// TIA Portal project "Laptrinhnangcaocuoiki_V16" (V16)

(* hardware
DEVICE "S7-1200 station_1"  S7-1200 Station
   slot 0: "Rack_0"  S7-1200 Rack  Rack  V1.0
   slot 1: "PLC_1"  CPU 1214C DC/DC/Rly  6ES7 214-1HG40-0XB0  V4.2
DEVICE "PC-System_1"  SIMATIC PC station
   slot 0: "SIMATIC PC station"  Rail  SIMATIC PC-Station  V1.0
      slot 125: "Stationmanager"  Station_Manager  V6.0.4
   slot 1: "HMI_RT_1"  WinCC RT Advanced  6AV2 104-0xxxx-xxxx  15.0.0.0
      slot 33792: "Host interface"  Host interface
   slot 2: "IE general_1"  IE General  IE_CP  V8.2.0
*)

// ===== PLC "PLC_1"  CPU 1214C DC/DC/Rly =====

VAR_GLOBAL   // PLC tag table "Default tag table"
   "Clock_Byte" AT %MB100 : Byte;
   "Clock_10Hz" AT %M100.0 : Bool;
   "Clock_5Hz" AT %M100.1 : Bool;
   "Clock_2.5Hz" AT %M100.2 : Bool;
   "Clock_2Hz" AT %M100.3 : Bool;
   "Clock_1.25Hz" AT %M100.4 : Bool;
   "Clock_1Hz" AT %M100.5 : Bool;
   "Clock_0.625Hz" AT %M100.6 : Bool;
   "Clock_0.5Hz" AT %M100.7 : Bool;
   "Tag_6" AT %M20.0 : Bool;
   "Tag_7" AT %M20.1 : Bool;
   "Tag_14" AT %M20.2 : Bool;
   "Tag_17" AT %M20.3 : Bool;
   "Tag_18" AT %M20.4 : Bool;
   "Tag_24" AT %M20.5 : Bool;
   "Tag_32" AT %M20.6 : Bool;
   "Tag_33" AT %M20.7 : Bool;
   "Tag_34" AT %M21.0 : Bool;
   "Tag_35" AT %M21.1 : Bool;
   "Tag_1" AT %M21.2 : Bool;
   "Tag_36" AT %M21.3 : Bool;
   "Tag_37" AT %M21.4 : Bool;
   "Tag_38" AT %M21.5 : Bool;
   "Tag_39" AT %M21.6 : Bool;
   "Tag_40" AT %M21.7 : Bool;
   "Tag_41" AT %M22.0 : Bool;
   "Tag_42" AT %M22.2 : Bool;
   "Tag_43" AT %M22.1 : Bool;
   "Tag_44" AT %M22.3 : Bool;
   "Tag_45" AT %M22.4 : Bool;
   "Tag_46" AT %M22.5 : Bool;
   "Tag_47" AT %M22.6 : Bool;
   "Tag_48" AT %M22.7 : Bool;
   "Tag_49" AT %M23.0 : Bool;
   "Tag_50" AT %M23.1 : Bool;
   "Tag_51" AT %M23.2 : Bool;
   "Tag_52" AT %M23.3 : Bool;
   "Tag_53" AT %M23.4 : Bool;
   "Tag_54" AT %M23.5 : Bool;
   "Tag_55" AT %M23.6 : Bool;
   "Tag_56" AT %M23.7 : Bool;
   "Tag_57" AT %M24.0 : Bool;
   "Tag_58" AT %M24.1 : Bool;
   "Tag_59" AT %M24.2 : Bool;
   "Tag_2" AT %M24.3 : Bool;
   "Tag_3" AT %M24.4 : Bool;
   "Tag_4" AT %M24.5 : Bool;
   "Tag_5" AT %M24.6 : Bool;
   "Tag_8" AT %M24.7 : Bool;
   "Tag_9" AT %M25.0 : Bool;
   "Tag_10" AT %M25.1 : Bool;
   "Tag_11" AT %M25.2 : Bool;
   "Tag_12" AT %M25.3 : Bool;
   "Tag_13" AT %M25.4 : Bool;
   "Tag_15" AT %M25.5 : Bool;
   "Tag_16" AT %M25.6 : Bool;
   "Tag_19" AT %M25.7 : Bool;
   "Tag_20" AT %M26.0 : Bool;
   "Tag_21" AT %M26.1 : Bool;
   "Tag_22" AT %M26.2 : Bool;
   "Tag_23" AT %M26.3 : Bool;
   "Tag_25" AT %M26.4 : Bool;
   "Tag_26" AT %M26.5 : Bool;
   "Tag_27" AT %M26.6 : Bool;
   "Tag_28" AT %M26.7 : Bool;
   "Tag_29" AT %M27.0 : Bool;
   "Tag_30" AT %M27.1 : Bool;
   "Tag_31" AT %M27.2 : Bool;
   "Tag_60" AT %M27.3 : Bool;
   "Tag_61" AT %M27.4 : Bool;
   "Tag_62" AT %M27.5 : Bool;
   "Tag_63" AT %M27.7 : Bool;
   "Tag_64" AT %M27.6 : Bool;
   "Tag_65" AT %M28.0 : Bool;
   "Tag_66" AT %M28.1 : Bool;
   "Tag_67" AT %M28.2 : Bool;
   "Tag_68" AT %M28.3 : Bool;
   "Tag_69" AT %M28.4 : Bool;
   "Tag_70" AT %M28.5 : Bool;
   "Tag_71" AT %M28.6 : Bool;
   "Tag_72" AT %M28.7 : Bool;
   "Tag_73" AT %M29.0 : Bool;
   "Tag_74" AT %M29.1 : Bool;
   "Tag_75" AT %M29.2 : Bool;
   "Tag_76" AT %M29.3 : Bool;
   "Tag_77" AT %M29.4 : Bool;
   "Tag_78" AT %M29.5 : Bool;
   "Tag_79" AT %M29.6 : Bool;
   "Tag_80" AT %M29.7 : Bool;
   "Tag_81" AT %M30.1 : Bool;
   "Tag_82" AT %M30.2 : Bool;
   "Tag_83" AT %M30.0 : Bool;
   "Tag_84" AT %M30.3 : Bool;
   "Tag_85" AT %M30.4 : Bool;
   "Tag_86" AT %M30.5 : Bool;
   "Tag_87" AT %M30.6 : Bool;
   "Tag_88" AT %M30.7 : Bool;
   "Tag_89" AT %M31.0 : Bool;
   "Tag_90" AT %M31.1 : Bool;
   "Tag_91" AT %M31.2 : Bool;
END_VAR

VAR_GLOBAL   // PLC tag table "M_tag"
   "mStart" AT %M0.0 : Bool;
   "mStop" AT %M0.1 : Bool;
   "mControlOn" AT %M0.2 : Bool;
   "mEnableXiloRice" AT %M0.3 : Bool;
   "mEnableXiloCorn" AT %M0.6 : Bool;
   "mEnableXiloCassava" AT %M1.2 : Bool;
   "mEnableXiloBean" AT %M1.4 : Bool;
   "mEnableXiloFish" AT %M1.7 : Bool;
   "mEnablePourToScale1" AT %M2.6 : Bool;
   "mEnableInverter1_10Hz" AT %M2.7 : Bool;
   "mEnableInverter1_5Hz" AT %M3.0 : Bool;
   "mEnableInverter1_1Hz" AT %M3.1 : Bool;
   "mEnableXiloRice1" AT %M0.4 : Bool;
   "mEnableXiloRice2" AT %M0.5 : Bool;
   "mEnableXiloRice3" AT %M0.7 : Bool;
   "mEnableXiloCorn4" AT %M1.0 : Bool;
   "mEnableXiloCorn5" AT %M1.1 : Bool;
   "mEnableXiloCorn6" AT %M1.3 : Bool;
   "mEnableXiloCorn7" AT %M1.5 : Bool;
   "mEnableXiloCassava8" AT %M1.6 : Bool;
   "mEnableXiloCassava9" AT %M2.0 : Bool;
   "mEnablePourToScale2" AT %M3.2 : Bool;
   "mEnableInverter2_10Hz" AT %M3.3 : Bool;
   "mEnableInverter2_5Hz" AT %M3.4 : Bool;
   "mEnableInverter2_1Hz" AT %M3.5 : Bool;
   "mEnableXiloBean10" AT %M2.1 : Bool;
   "mEnableXiloBean11" AT %M2.2 : Bool;
   "mEnableXiloBean12" AT %M3.6 : Bool;
   "mEnableXiloFish13" AT %M3.7 : Bool;
   "mEnableXiloFish14" AT %M4.0 : Bool;
   "mEnableXiloFish15" AT %M4.1 : Bool;
   "mEnableXiloFish16" AT %M4.2 : Bool;
   "mEnableMotorMixTank" AT %M4.3 : Bool;
   "mEnableValveScale1" AT %M4.4 : Bool;
   "mEnableValveScale2" AT %M4.5 : Bool;
   "mDisableMotorMixTank" AT %M4.7 : Bool;
   "mEnableValveMixTank" AT %M4.6 : Bool;
   "mEnablePourMixTank" AT %M5.2 : Bool;
END_VAR

VAR_GLOBAL   // PLC tag table "Q_tag"
   "qXiloRice1" AT %Q0.0 : Bool;
   "qXiloRice2" AT %Q0.1 : Bool;
   "qXiloRice3" AT %Q0.2 : Bool;
   "qXiloCorn4" AT %Q0.3 : Bool;
   "qXiloCorn5" AT %Q0.4 : Bool;
   "qXiloCorn6" AT %Q0.5 : Bool;
   "qXiloCorn7" AT %Q0.6 : Bool;
   "qXiloCassava8" AT %Q0.7 : Bool;
   "qXiloCassava9" AT %Q1.0 : Bool;
   "qXiloBean10" AT %Q1.1 : Bool;
   "qXiloBean11" AT %Q1.2 : Bool;
   "qXiloBean12" AT %Q1.3 : Bool;
   "qXiloFish13" AT %Q1.4 : Bool;
   "qXiloFish14" AT %Q1.5 : Bool;
   "qXiloFish15" AT %Q1.6 : Bool;
   "qXiloFish16" AT %Q1.7 : Bool;
   "qValveScale1" AT %Q2.0 : Bool;
   "qValveScale2" AT %Q2.1 : Bool;
   "qMotorMixTank" AT %Q2.2 : Bool;
   "qValveMixTank" AT %Q2.3 : Bool;
END_VAR

VAR_GLOBAL   // PLC tag table "mSensor"
   "mSensorHightXilo1" AT %M10.0 : Bool;
   "mSensorHightXilo2" AT %M10.1 : Bool;
   "mSensorHightXilo3" AT %M10.2 : Bool;
   "mSensorHightXilo4" AT %M10.3 : Bool;
   "mSensorHightXilo5" AT %M10.4 : Bool;
   "mSensorHightXilo6" AT %M10.5 : Bool;
   "mSensorHightXilo7" AT %M10.6 : Bool;
   "mSensorHightXilo8" AT %M10.7 : Bool;
   "mSensorHightXilo9" AT %M11.0 : Bool;
   "mSensorHightXilo10" AT %M11.1 : Bool;
   "mSensorHightXilo11" AT %M11.2 : Bool;
   "mSensorHightXilo12" AT %M11.3 : Bool;
   "mSensorHightXilo13" AT %M11.4 : Bool;
   "mSensorHightXilo14" AT %M11.5 : Bool;
   "mSensorHightXilo15" AT %M11.6 : Bool;
   "mSensorHightXilo16" AT %M11.7 : Bool;
   "mSensorLowXilo1" AT %M12.0 : Bool;
   "mSensorLowXilo2" AT %M12.1 : Bool;
   "mSensorLowXilo3" AT %M12.2 : Bool;
   "mSensorLowXilo4" AT %M12.3 : Bool;
   "mSensorLowXilo5" AT %M12.4 : Bool;
   "mSensorLowXilo6" AT %M12.5 : Bool;
   "mSensorLowXilo7" AT %M12.6 : Bool;
   "mSensorLowXilo8" AT %M12.7 : Bool;
   "mSensorLowXilo9" AT %M13.0 : Bool;
   "mSensorLowXilo10" AT %M13.1 : Bool;
   "mSensorLowXilo11" AT %M13.2 : Bool;
   "mSensorLowXilo12" AT %M13.3 : Bool;
   "mSensorLowXilo13" AT %M13.4 : Bool;
   "mSensorLowXilo14" AT %M13.5 : Bool;
   "mSensorLowXilo15" AT %M13.6 : Bool;
   "mSensorLowXilo16" AT %M13.7 : Bool;
   "mSensorValveScale1" AT %M2.3 : Bool;
   "mSensorValveScale2" AT %M2.4 : Bool;
   "mSensorMixTankHight" AT %M2.5 : Bool;
   "mSensorMixTankLow" AT %M5.0 : Bool;
   "mSensorValveMixTank" AT %M5.1 : Bool;
END_VAR

DATA_BLOCK "Data_block_1"   // DB1
{ S7_Optimized_Access := 'FALSE' }
VERSION : 0.1
   VAR
      "Missing Rice" : Real;
      "Missing Corn" : Real;
      "Missing Cassava" : Real;
      "Missing Bean" : Real;
      "Missing Fish" : Real;
      "Act Scale 1" : Real;
      "Act Scale 2" : Real;
      "Set Scale 1" : Real := 0.0001;
      "Set Scale 2" : Real := 0.0001;
      "Ratio Scale 1" : Real;
      "Ratio Scale 2" : Real;
      "Set Each Xilo Rice" : Real;
      "Set Each Xilo Corn" : Real;
      "Set Each Xilo Cassava" : Real;
      "Accumulate Scale 1" : Real := 0.0;
      "Accumulate Scale 2" : Real;
      "Set Each Xilo Bean" : Real;
      "Set Each Xilo Fish" : Real;
   END_VAR
BEGIN
END_DATA_BLOCK

DATA_BLOCK "Data_block_2"   // DB3
{ S7_Optimized_Access := 'FALSE' }
VERSION : 0.1
   VAR
      "Input Rice" : Real := 0.0;
      "Input Corn" : Real := 0.0;
      "Input Cassava" : Real := 0.0;
      "Input Bean" : Real := 0.0;
      "Input Fish" : Real := 0.0;
      "Set Timer Mix" : Time := T#10s;
   END_VAR
BEGIN
END_DATA_BLOCK

DATA_BLOCK "Data_block_3"   // DB4
{ S7_Optimized_Access := 'FALSE' }
VERSION : 0.1
   VAR
      ActScale1 : Real;
      ActScale2 : Real;
      ActTimerMix : Time := T#0Ms;
   END_VAR
BEGIN
END_DATA_BLOCK

// folder: System blocks/Program resources

DATA_BLOCK "IEC_Timer_0_DB"   // DB2
{ S7_Optimized_Access := 'TRUE' }
AUTHOR : Simatic
FAMILY : IEC
NAME : IEC_TMR
VERSION : 1.0
// stored: InstanceOfName IEC_TIMER
"IEC_TIMER"
BEGIN
END_DATA_BLOCK

// folder: (top level)

FUNCTION "Select_Xilo_Scale1" : Void   // FC1, LAD
{ S7_Optimized_Access := 'TRUE' }
VERSION : 0.1
   VAR_TEMP   // added for the SCL form of the ladder/FBD networks
      _w1 : Bool;
      _w2 : Bool;
      _w3 : Bool;
   END_VAR
BEGIN

REGION Network 1
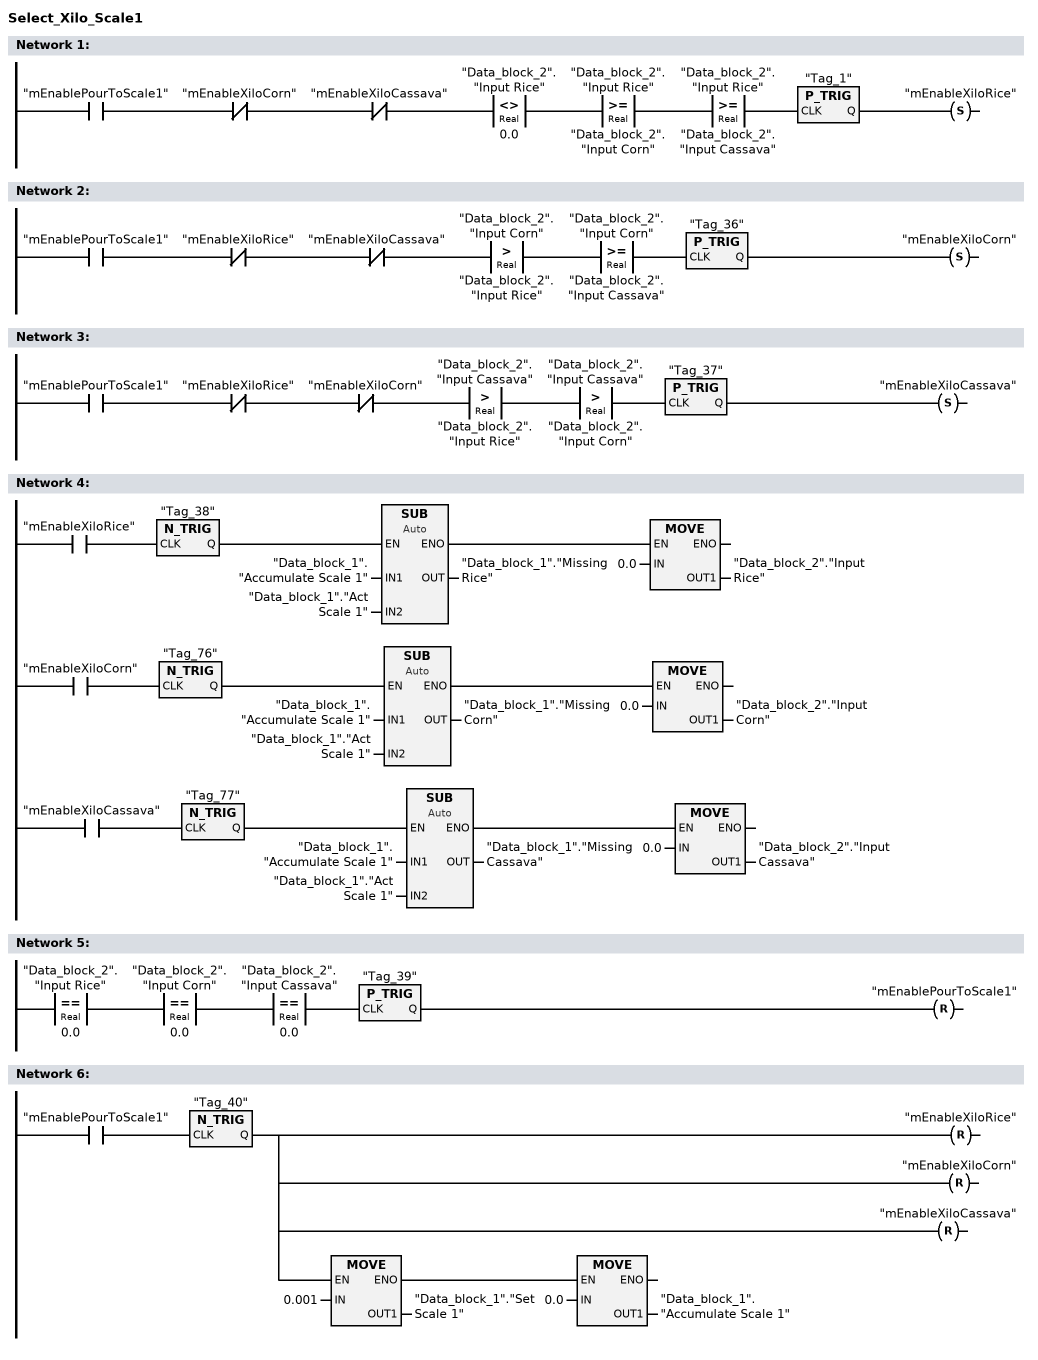
   RUNG wire#powerrail
      Contact( "mEnablePourToScale1" )
      I_Contact( "mEnableXiloCorn" )
      I_Contact( "mEnableXiloCassava" )
      { S7_Templates := "SrcType := Real" } NE_Contact(in1 := "Data_block_2"."Input Rice", in2 := 0.0)
      { S7_Templates := "SrcType := Real" } GE_Contact(in1 := "Data_block_2"."Input Rice", in2 := "Data_block_2"."Input Corn")
      { S7_Templates := "SrcType := Real" } GE_Contact(in1 := "Data_block_2"."Input Rice", in2 := "Data_block_2"."Input Cassava")
      P_Trig( "Tag_1" )
      S_Coil( "mEnableXiloRice" )
   END_RUNG
   // the same network as SCL:
   #_w1 := "mEnablePourToScale1" AND NOT "mEnableXiloCorn" AND NOT "mEnableXiloCassava" AND ("Data_block_2"."Input Rice" <> 0.0) AND ("Data_block_2"."Input Rice" >= "Data_block_2"."Input Corn") AND ("Data_block_2"."Input Rice" >= "Data_block_2"."Input Cassava");
   #_w2 := #_w1 AND NOT "Tag_1";   // rising edge
   "Tag_1" := #_w1;
   IF #_w2 THEN "mEnableXiloRice" := TRUE; END_IF;
END_REGION

REGION Network 2
   RUNG wire#powerrail
      Contact( "mEnablePourToScale1" )
      I_Contact( "mEnableXiloRice" )
      I_Contact( "mEnableXiloCassava" )
      { S7_Templates := "SrcType := Real" } GT_Contact(in1 := "Data_block_2"."Input Corn", in2 := "Data_block_2"."Input Rice")
      { S7_Templates := "SrcType := Real" } GE_Contact(in1 := "Data_block_2"."Input Corn", in2 := "Data_block_2"."Input Cassava")
      P_Trig( "Tag_36" )
      S_Coil( "mEnableXiloCorn" )
   END_RUNG
   // the same network as SCL:
   #_w1 := "mEnablePourToScale1" AND NOT "mEnableXiloRice" AND NOT "mEnableXiloCassava" AND ("Data_block_2"."Input Corn" > "Data_block_2"."Input Rice") AND ("Data_block_2"."Input Corn" >= "Data_block_2"."Input Cassava");
   #_w2 := #_w1 AND NOT "Tag_36";   // rising edge
   "Tag_36" := #_w1;
   IF #_w2 THEN "mEnableXiloCorn" := TRUE; END_IF;
END_REGION

REGION Network 3
   RUNG wire#powerrail
      Contact( "mEnablePourToScale1" )
      I_Contact( "mEnableXiloRice" )
      I_Contact( "mEnableXiloCorn" )
      { S7_Templates := "SrcType := Real" } GT_Contact(in1 := "Data_block_2"."Input Cassava", in2 := "Data_block_2"."Input Rice")
      { S7_Templates := "SrcType := Real" } GT_Contact(in1 := "Data_block_2"."Input Cassava", in2 := "Data_block_2"."Input Corn")
      P_Trig( "Tag_37" )
      S_Coil( "mEnableXiloCassava" )
   END_RUNG
   // the same network as SCL:
   #_w1 := "mEnablePourToScale1" AND NOT "mEnableXiloRice" AND NOT "mEnableXiloCorn" AND ("Data_block_2"."Input Cassava" > "Data_block_2"."Input Rice") AND ("Data_block_2"."Input Cassava" > "Data_block_2"."Input Corn");
   #_w2 := #_w1 AND NOT "Tag_37";   // rising edge
   "Tag_37" := #_w1;
   IF #_w2 THEN "mEnableXiloCassava" := TRUE; END_IF;
END_REGION

REGION Network 4
   RUNG wire#powerrail
      Contact( "mEnableXiloRice" )
      N_Trig( "Tag_38" )
      Sub(in1 := "Data_block_1"."Accumulate Scale 1", in2 := "Data_block_1"."Act Scale 1", out => "Data_block_1"."Missing Rice")
      Move(in := 0.0, out1 => "Data_block_2"."Input Rice")
   END_RUNG
   RUNG wire#powerrail
      Contact( "mEnableXiloCorn" )
      N_Trig( "Tag_76" )
      Sub(in1 := "Data_block_1"."Accumulate Scale 1", in2 := "Data_block_1"."Act Scale 1", out => "Data_block_1"."Missing Corn")
      Move(in := 0.0, out1 => "Data_block_2"."Input Corn")
   END_RUNG
   RUNG wire#powerrail
      Contact( "mEnableXiloCassava" )
      N_Trig( "Tag_77" )
      Sub(in1 := "Data_block_1"."Accumulate Scale 1", in2 := "Data_block_1"."Act Scale 1", out => "Data_block_1"."Missing Cassava")
      Move(in := 0.0, out1 => "Data_block_2"."Input Cassava")
   END_RUNG
   // the same network as SCL:
   #_w1 := NOT "mEnableXiloRice" AND "Tag_38";   // falling edge
   "Tag_38" := "mEnableXiloRice";
   IF #_w1 THEN
       "Data_block_1"."Missing Rice" := "Data_block_1"."Accumulate Scale 1" - "Data_block_1"."Act Scale 1";
       "Data_block_2"."Input Rice" := 0.0;
   END_IF;
   #_w2 := NOT "mEnableXiloCorn" AND "Tag_76";   // falling edge
   "Tag_76" := "mEnableXiloCorn";
   IF #_w2 THEN
       "Data_block_1"."Missing Corn" := "Data_block_1"."Accumulate Scale 1" - "Data_block_1"."Act Scale 1";
       "Data_block_2"."Input Corn" := 0.0;
   END_IF;
   #_w3 := NOT "mEnableXiloCassava" AND "Tag_77";   // falling edge
   "Tag_77" := "mEnableXiloCassava";
   IF #_w3 THEN
       "Data_block_1"."Missing Cassava" := "Data_block_1"."Accumulate Scale 1" - "Data_block_1"."Act Scale 1";
       "Data_block_2"."Input Cassava" := 0.0;
   END_IF;
END_REGION

REGION Network 5
   RUNG wire#powerrail
      { S7_Templates := "SrcType := Real" } EQ_Contact(in1 := "Data_block_2"."Input Rice", in2 := 0.0)
      { S7_Templates := "SrcType := Real" } EQ_Contact(in1 := "Data_block_2"."Input Corn", in2 := 0.0)
      { S7_Templates := "SrcType := Real" } EQ_Contact(in1 := "Data_block_2"."Input Cassava", in2 := 0.0)
      P_Trig( "Tag_39" )
      R_Coil( "mEnablePourToScale1" )
   END_RUNG
   // the same network as SCL:
   #_w1 := ("Data_block_2"."Input Rice" = 0.0) AND ("Data_block_2"."Input Corn" = 0.0) AND ("Data_block_2"."Input Cassava" = 0.0);
   #_w2 := #_w1 AND NOT "Tag_39";   // rising edge
   "Tag_39" := #_w1;
   IF #_w2 THEN "mEnablePourToScale1" := FALSE; END_IF;
END_REGION

REGION Network 6
   RUNG wire#powerrail
      Contact( "mEnablePourToScale1" )
      N_Trig( "Tag_40" )
      wire#w1
      R_Coil( "mEnableXiloRice" )
   END_RUNG
   RUNG wire#w1
      R_Coil( "mEnableXiloCorn" )
   END_RUNG
   RUNG wire#w1
      R_Coil( "mEnableXiloCassava" )
   END_RUNG
   RUNG wire#w1
      Move(in := 0.001, out1 => "Data_block_1"."Set Scale 1")
      Move(in := 0.0, out1 => "Data_block_1"."Accumulate Scale 1")
   END_RUNG
   // the same network as SCL:
   #_w1 := NOT "mEnablePourToScale1" AND "Tag_40";   // falling edge
   "Tag_40" := "mEnablePourToScale1";
   IF #_w1 THEN
       "mEnableXiloRice" := FALSE;
       "mEnableXiloCorn" := FALSE;
       "mEnableXiloCassava" := FALSE;
       "Data_block_1"."Set Scale 1" := 0.001;
       "Data_block_1"."Accumulate Scale 1" := 0.0;
   END_IF;
END_REGION
END_FUNCTION

FUNCTION "Add_Value_Weight" : Void   // FC2, LAD
{ S7_Optimized_Access := 'TRUE' }
VERSION : 0.1
   VAR_TEMP   // added for the SCL form of the ladder/FBD networks
      _w1 : Bool;
      _w2 : Bool;
      _w3 : Bool;
      _w4 : Bool;
   END_VAR
BEGIN

REGION Network 1
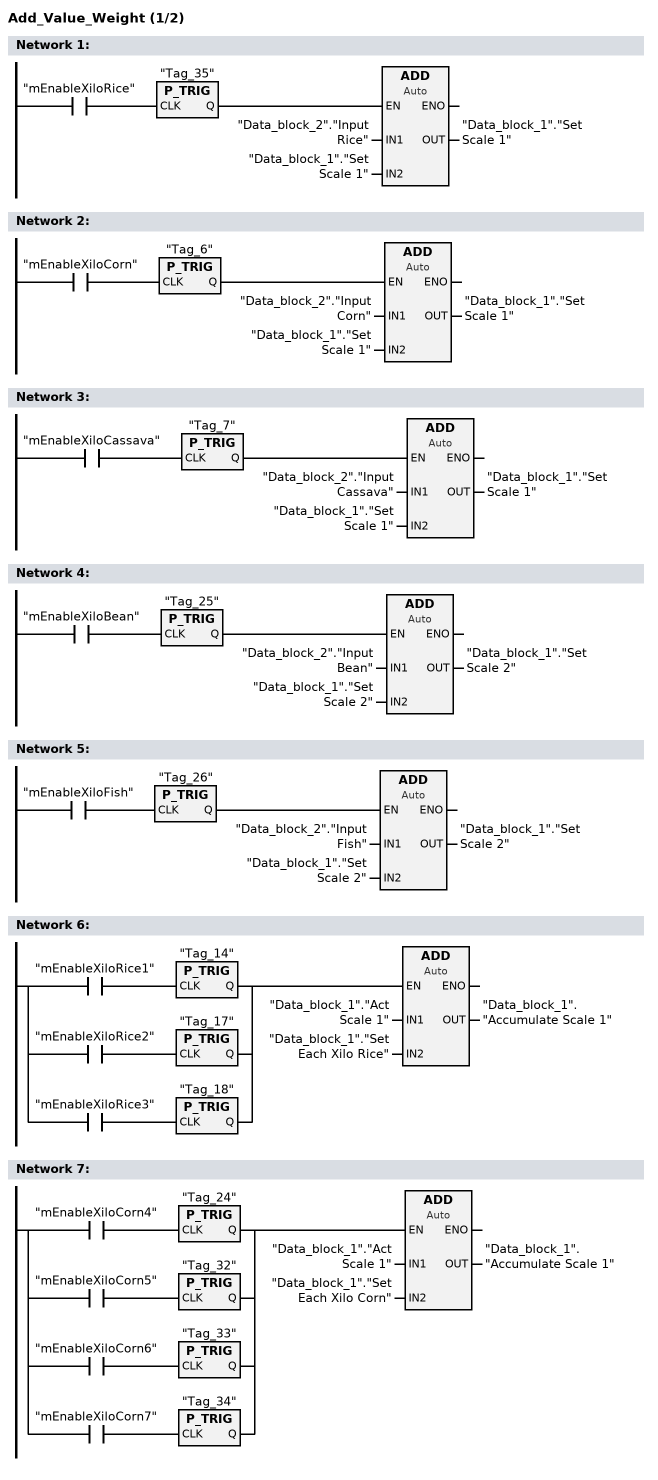
   RUNG wire#powerrail
      Contact( "mEnableXiloRice" )
      P_Trig( "Tag_35" )
      Add(in1 := "Data_block_2"."Input Rice", in2 := "Data_block_1"."Set Scale 1", out => "Data_block_1"."Set Scale 1")
   END_RUNG
   // the same network as SCL:
   #_w1 := "mEnableXiloRice" AND NOT "Tag_35";   // rising edge
   "Tag_35" := "mEnableXiloRice";
   IF #_w1 THEN
       "Data_block_1"."Set Scale 1" := "Data_block_2"."Input Rice" + "Data_block_1"."Set Scale 1";
   END_IF;
END_REGION

REGION Network 2
   RUNG wire#powerrail
      Contact( "mEnableXiloCorn" )
      P_Trig( "Tag_6" )
      Add(in1 := "Data_block_2"."Input Corn", in2 := "Data_block_1"."Set Scale 1", out => "Data_block_1"."Set Scale 1")
   END_RUNG
   // the same network as SCL:
   #_w1 := "mEnableXiloCorn" AND NOT "Tag_6";   // rising edge
   "Tag_6" := "mEnableXiloCorn";
   IF #_w1 THEN
       "Data_block_1"."Set Scale 1" := "Data_block_2"."Input Corn" + "Data_block_1"."Set Scale 1";
   END_IF;
END_REGION

REGION Network 3
   RUNG wire#powerrail
      Contact( "mEnableXiloCassava" )
      P_Trig( "Tag_7" )
      Add(in1 := "Data_block_2"."Input Cassava", in2 := "Data_block_1"."Set Scale 1", out => "Data_block_1"."Set Scale 1")
   END_RUNG
   // the same network as SCL:
   #_w1 := "mEnableXiloCassava" AND NOT "Tag_7";   // rising edge
   "Tag_7" := "mEnableXiloCassava";
   IF #_w1 THEN
       "Data_block_1"."Set Scale 1" := "Data_block_2"."Input Cassava" + "Data_block_1"."Set Scale 1";
   END_IF;
END_REGION

REGION Network 4
   RUNG wire#powerrail
      Contact( "mEnableXiloBean" )
      P_Trig( "Tag_25" )
      Add(in1 := "Data_block_2"."Input Bean", in2 := "Data_block_1"."Set Scale 2", out => "Data_block_1"."Set Scale 2")
   END_RUNG
   // the same network as SCL:
   #_w1 := "mEnableXiloBean" AND NOT "Tag_25";   // rising edge
   "Tag_25" := "mEnableXiloBean";
   IF #_w1 THEN
       "Data_block_1"."Set Scale 2" := "Data_block_2"."Input Bean" + "Data_block_1"."Set Scale 2";
   END_IF;
END_REGION

REGION Network 5
   RUNG wire#powerrail
      Contact( "mEnableXiloFish" )
      P_Trig( "Tag_26" )
      Add(in1 := "Data_block_2"."Input Fish", in2 := "Data_block_1"."Set Scale 2", out => "Data_block_1"."Set Scale 2")
   END_RUNG
   // the same network as SCL:
   #_w1 := "mEnableXiloFish" AND NOT "Tag_26";   // rising edge
   "Tag_26" := "mEnableXiloFish";
   IF #_w1 THEN
       "Data_block_1"."Set Scale 2" := "Data_block_2"."Input Fish" + "Data_block_1"."Set Scale 2";
   END_IF;
END_REGION

REGION Network 6
   RUNG wire#powerrail
      Contact( "mEnableXiloRice1" )
      P_Trig( "Tag_14" )
      wire#w1
      Add(in1 := "Data_block_1"."Act Scale 1", in2 := "Data_block_1"."Set Each Xilo Rice", out => "Data_block_1"."Accumulate Scale 1")
   END_RUNG
   RUNG wire#powerrail
      Contact( "mEnableXiloRice2" )
      P_Trig( "Tag_17" )
   END_RUNG wire#w1
   RUNG wire#powerrail
      Contact( "mEnableXiloRice3" )
      P_Trig( "Tag_18" )
   END_RUNG wire#w1
   // the same network as SCL:
   #_w1 := "mEnableXiloRice1" AND NOT "Tag_14";   // rising edge
   "Tag_14" := "mEnableXiloRice1";
   #_w2 := "mEnableXiloRice2" AND NOT "Tag_17";   // rising edge
   "Tag_17" := "mEnableXiloRice2";
   #_w3 := "mEnableXiloRice3" AND NOT "Tag_18";   // rising edge
   "Tag_18" := "mEnableXiloRice3";
   IF #_w1 OR #_w2 OR #_w3 THEN
       "Data_block_1"."Accumulate Scale 1" := "Data_block_1"."Act Scale 1" + "Data_block_1"."Set Each Xilo Rice";
   END_IF;
END_REGION

REGION Network 7
   RUNG wire#powerrail
      Contact( "mEnableXiloCorn4" )
      P_Trig( "Tag_24" )
      wire#w1
      Add(in1 := "Data_block_1"."Act Scale 1", in2 := "Data_block_1"."Set Each Xilo Corn", out => "Data_block_1"."Accumulate Scale 1")
   END_RUNG
   RUNG wire#powerrail
      Contact( "mEnableXiloCorn5" )
      P_Trig( "Tag_32" )
   END_RUNG wire#w1
   RUNG wire#powerrail
      Contact( "mEnableXiloCorn6" )
      P_Trig( "Tag_33" )
   END_RUNG wire#w1
   RUNG wire#powerrail
      Contact( "mEnableXiloCorn7" )
      P_Trig( "Tag_34" )
   END_RUNG wire#w1
   // the same network as SCL:
   #_w1 := "mEnableXiloCorn4" AND NOT "Tag_24";   // rising edge
   "Tag_24" := "mEnableXiloCorn4";
   #_w2 := "mEnableXiloCorn5" AND NOT "Tag_32";   // rising edge
   "Tag_32" := "mEnableXiloCorn5";
   #_w3 := "mEnableXiloCorn6" AND NOT "Tag_33";   // rising edge
   "Tag_33" := "mEnableXiloCorn6";
   #_w4 := "mEnableXiloCorn7" AND NOT "Tag_34";   // rising edge
   "Tag_34" := "mEnableXiloCorn7";
   IF #_w1 OR #_w2 OR #_w3 OR #_w4 THEN
       "Data_block_1"."Accumulate Scale 1" := "Data_block_1"."Act Scale 1" + "Data_block_1"."Set Each Xilo Corn";
   END_IF;
END_REGION

REGION Network 8
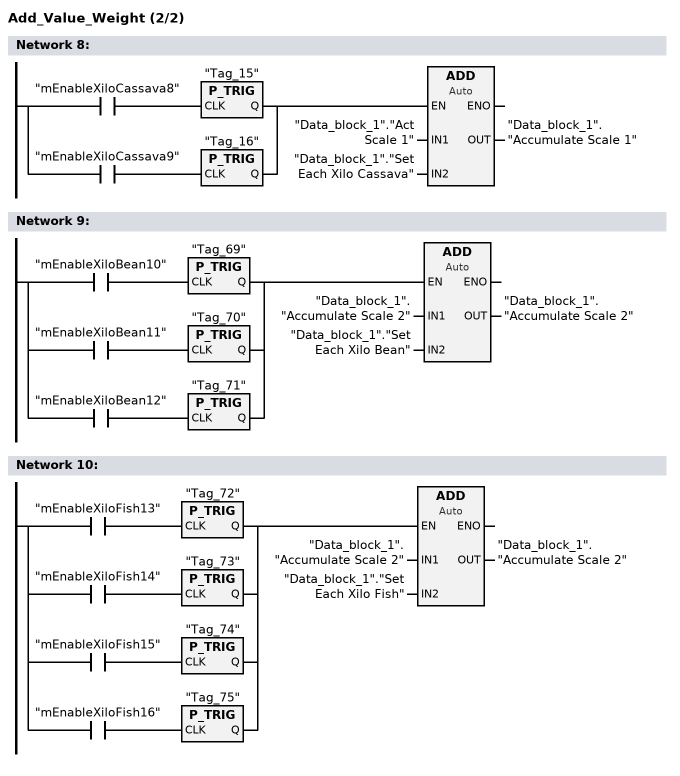
   RUNG wire#powerrail
      Contact( "mEnableXiloCassava8" )
      P_Trig( "Tag_15" )
      wire#w1
      Add(in1 := "Data_block_1"."Act Scale 1", in2 := "Data_block_1"."Set Each Xilo Cassava", out => "Data_block_1"."Accumulate Scale 1")
   END_RUNG
   RUNG wire#powerrail
      Contact( "mEnableXiloCassava9" )
      P_Trig( "Tag_16" )
   END_RUNG wire#w1
   // the same network as SCL:
   #_w1 := "mEnableXiloCassava8" AND NOT "Tag_15";   // rising edge
   "Tag_15" := "mEnableXiloCassava8";
   #_w2 := "mEnableXiloCassava9" AND NOT "Tag_16";   // rising edge
   "Tag_16" := "mEnableXiloCassava9";
   IF #_w1 OR #_w2 THEN
       "Data_block_1"."Accumulate Scale 1" := "Data_block_1"."Act Scale 1" + "Data_block_1"."Set Each Xilo Cassava";
   END_IF;
END_REGION

REGION Network 9
   RUNG wire#powerrail
      Contact( "mEnableXiloBean10" )
      P_Trig( "Tag_69" )
      wire#w1
      Add(in1 := "Data_block_1"."Accumulate Scale 2", in2 := "Data_block_1"."Set Each Xilo Bean", out => "Data_block_1"."Accumulate Scale 2")
   END_RUNG
   RUNG wire#powerrail
      Contact( "mEnableXiloBean11" )
      P_Trig( "Tag_70" )
   END_RUNG wire#w1
   RUNG wire#powerrail
      Contact( "mEnableXiloBean12" )
      P_Trig( "Tag_71" )
   END_RUNG wire#w1
   // the same network as SCL:
   #_w1 := "mEnableXiloBean10" AND NOT "Tag_69";   // rising edge
   "Tag_69" := "mEnableXiloBean10";
   #_w2 := "mEnableXiloBean11" AND NOT "Tag_70";   // rising edge
   "Tag_70" := "mEnableXiloBean11";
   #_w3 := "mEnableXiloBean12" AND NOT "Tag_71";   // rising edge
   "Tag_71" := "mEnableXiloBean12";
   IF #_w1 OR #_w2 OR #_w3 THEN
       "Data_block_1"."Accumulate Scale 2" := "Data_block_1"."Accumulate Scale 2" + "Data_block_1"."Set Each Xilo Bean";
   END_IF;
END_REGION

REGION Network 10
   RUNG wire#powerrail
      Contact( "mEnableXiloFish13" )
      P_Trig( "Tag_72" )
      wire#w1
      Add(in1 := "Data_block_1"."Accumulate Scale 2", in2 := "Data_block_1"."Set Each Xilo Fish", out => "Data_block_1"."Accumulate Scale 2")
   END_RUNG
   RUNG wire#powerrail
      Contact( "mEnableXiloFish14" )
      P_Trig( "Tag_73" )
   END_RUNG wire#w1
   RUNG wire#powerrail
      Contact( "mEnableXiloFish15" )
      P_Trig( "Tag_74" )
   END_RUNG wire#w1
   RUNG wire#powerrail
      Contact( "mEnableXiloFish16" )
      P_Trig( "Tag_75" )
   END_RUNG wire#w1
   // the same network as SCL:
   #_w1 := "mEnableXiloFish13" AND NOT "Tag_72";   // rising edge
   "Tag_72" := "mEnableXiloFish13";
   #_w2 := "mEnableXiloFish14" AND NOT "Tag_73";   // rising edge
   "Tag_73" := "mEnableXiloFish14";
   #_w3 := "mEnableXiloFish15" AND NOT "Tag_74";   // rising edge
   "Tag_74" := "mEnableXiloFish15";
   #_w4 := "mEnableXiloFish16" AND NOT "Tag_75";   // rising edge
   "Tag_75" := "mEnableXiloFish16";
   IF #_w1 OR #_w2 OR #_w3 OR #_w4 THEN
       "Data_block_1"."Accumulate Scale 2" := "Data_block_1"."Accumulate Scale 2" + "Data_block_1"."Set Each Xilo Fish";
   END_IF;
END_REGION
END_FUNCTION

FUNCTION "SIMULINK_Act Scale" : Void   // FC3, LAD
{ S7_Optimized_Access := 'TRUE' }
VERSION : 0.1
   VAR_TEMP   // added for the SCL form of the ladder/FBD networks
      _w1 : Bool;
      _w2 : Bool;
   END_VAR
BEGIN

REGION Network 1
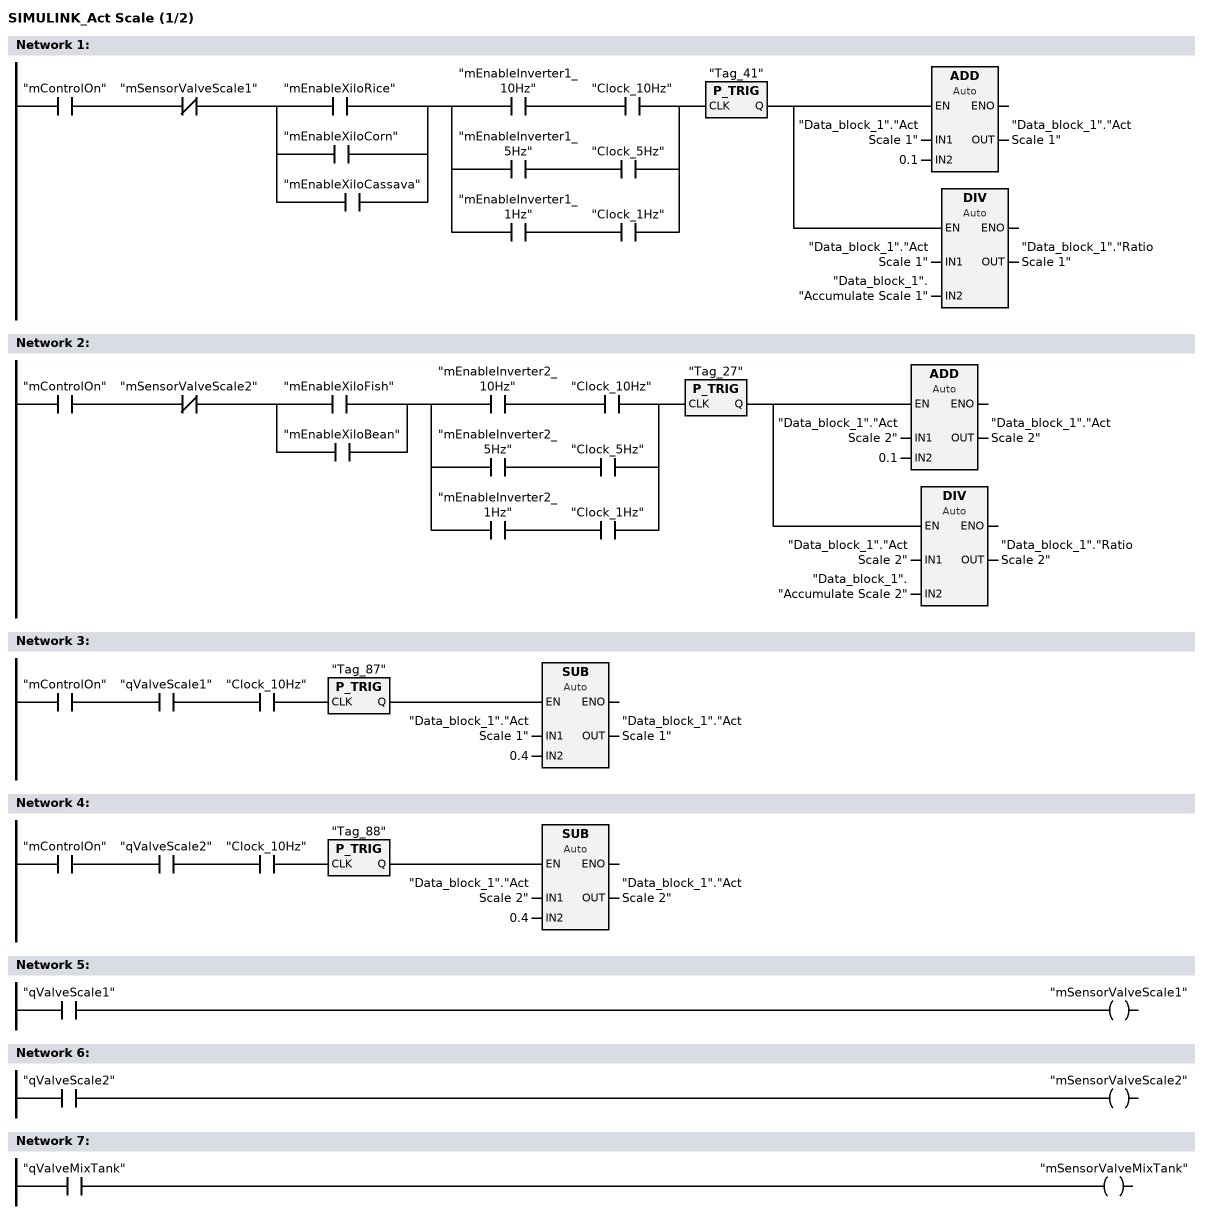
   RUNG wire#powerrail
      Contact( "mControlOn" )
      I_Contact( "mSensorValveScale1" )
      wire#w1
      Contact( "mEnableXiloRice" )
      wire#w2
      Contact( "mEnableInverter1_10Hz" )
      Contact( "Clock_10Hz" )
      wire#w3
      P_Trig( "Tag_41" )
      wire#w4
      Add(in1 := "Data_block_1"."Act Scale 1", in2 := 0.1, out => "Data_block_1"."Act Scale 1")
   END_RUNG
   RUNG wire#w1
      Contact( "mEnableXiloCorn" )
   END_RUNG wire#w2
   RUNG wire#w1
      Contact( "mEnableXiloCassava" )
   END_RUNG wire#w2
   RUNG wire#w2
      Contact( "mEnableInverter1_5Hz" )
      Contact( "Clock_5Hz" )
   END_RUNG wire#w3
   RUNG wire#w2
      Contact( "mEnableInverter1_1Hz" )
      Contact( "Clock_1Hz" )
   END_RUNG wire#w3
   RUNG wire#w4
      Div(in1 := "Data_block_1"."Act Scale 1", in2 := "Data_block_1"."Accumulate Scale 1", out => "Data_block_1"."Ratio Scale 1")
   END_RUNG
   // the same network as SCL:
   #_w1 := "mControlOn" AND NOT "mSensorValveScale1" AND ("mEnableXiloRice" OR "mEnableXiloCorn" OR "mEnableXiloCassava") AND (("mEnableInverter1_10Hz" AND "Clock_10Hz") OR ("mEnableInverter1_5Hz" AND "Clock_5Hz") OR ("mEnableInverter1_1Hz" AND "Clock_1Hz"));
   #_w2 := #_w1 AND NOT "Tag_41";   // rising edge
   "Tag_41" := #_w1;
   IF #_w2 THEN
       "Data_block_1"."Act Scale 1" := "Data_block_1"."Act Scale 1" + 0.1;
       "Data_block_1"."Ratio Scale 1" := "Data_block_1"."Act Scale 1" / "Data_block_1"."Accumulate Scale 1";
   END_IF;
END_REGION

REGION Network 2
   RUNG wire#powerrail
      Contact( "mControlOn" )
      I_Contact( "mSensorValveScale2" )
      wire#w1
      Contact( "mEnableXiloFish" )
      wire#w2
      Contact( "mEnableInverter2_10Hz" )
      Contact( "Clock_10Hz" )
      wire#w3
      P_Trig( "Tag_27" )
      wire#w4
      Add(in1 := "Data_block_1"."Act Scale 2", in2 := 0.1, out => "Data_block_1"."Act Scale 2")
   END_RUNG
   RUNG wire#w1
      Contact( "mEnableXiloBean" )
   END_RUNG wire#w2
   RUNG wire#w2
      Contact( "mEnableInverter2_5Hz" )
      Contact( "Clock_5Hz" )
   END_RUNG wire#w3
   RUNG wire#w2
      Contact( "mEnableInverter2_1Hz" )
      Contact( "Clock_1Hz" )
   END_RUNG wire#w3
   RUNG wire#w4
      Div(in1 := "Data_block_1"."Act Scale 2", in2 := "Data_block_1"."Accumulate Scale 2", out => "Data_block_1"."Ratio Scale 2")
   END_RUNG
   // the same network as SCL:
   #_w1 := "mControlOn" AND NOT "mSensorValveScale2" AND ("mEnableXiloFish" OR "mEnableXiloBean") AND (("mEnableInverter2_10Hz" AND "Clock_10Hz") OR ("mEnableInverter2_5Hz" AND "Clock_5Hz") OR ("mEnableInverter2_1Hz" AND "Clock_1Hz"));
   #_w2 := #_w1 AND NOT "Tag_27";   // rising edge
   "Tag_27" := #_w1;
   IF #_w2 THEN
       "Data_block_1"."Act Scale 2" := "Data_block_1"."Act Scale 2" + 0.1;
       "Data_block_1"."Ratio Scale 2" := "Data_block_1"."Act Scale 2" / "Data_block_1"."Accumulate Scale 2";
   END_IF;
END_REGION

REGION Network 3
   RUNG wire#powerrail
      Contact( "mControlOn" )
      Contact( "qValveScale1" )
      Contact( "Clock_10Hz" )
      P_Trig( "Tag_87" )
      Sub(in1 := "Data_block_1"."Act Scale 1", in2 := 0.4, out => "Data_block_1"."Act Scale 1")
   END_RUNG
   // the same network as SCL:
   #_w1 := "mControlOn" AND "qValveScale1" AND "Clock_10Hz";
   #_w2 := #_w1 AND NOT "Tag_87";   // rising edge
   "Tag_87" := #_w1;
   IF #_w2 THEN "Data_block_1"."Act Scale 1" := "Data_block_1"."Act Scale 1" - 0.4; END_IF;
END_REGION

REGION Network 4
   RUNG wire#powerrail
      Contact( "mControlOn" )
      Contact( "qValveScale2" )
      Contact( "Clock_10Hz" )
      P_Trig( "Tag_88" )
      Sub(in1 := "Data_block_1"."Act Scale 2", in2 := 0.4, out => "Data_block_1"."Act Scale 2")
   END_RUNG
   // the same network as SCL:
   #_w1 := "mControlOn" AND "qValveScale2" AND "Clock_10Hz";
   #_w2 := #_w1 AND NOT "Tag_88";   // rising edge
   "Tag_88" := #_w1;
   IF #_w2 THEN "Data_block_1"."Act Scale 2" := "Data_block_1"."Act Scale 2" - 0.4; END_IF;
END_REGION

REGION Network 5
   RUNG wire#powerrail
      Contact( "qValveScale1" )
      Coil( "mSensorValveScale1" )
   END_RUNG
   // the same network as SCL:
   "mSensorValveScale1" := "qValveScale1";
END_REGION

REGION Network 6
   RUNG wire#powerrail
      Contact( "qValveScale2" )
      Coil( "mSensorValveScale2" )
   END_RUNG
   // the same network as SCL:
   "mSensorValveScale2" := "qValveScale2";
END_REGION

REGION Network 7
   RUNG wire#powerrail
      Contact( "qValveMixTank" )
      Coil( "mSensorValveMixTank" )
   END_RUNG
   // the same network as SCL:
   "mSensorValveMixTank" := "qValveMixTank";
END_REGION

REGION Network 8
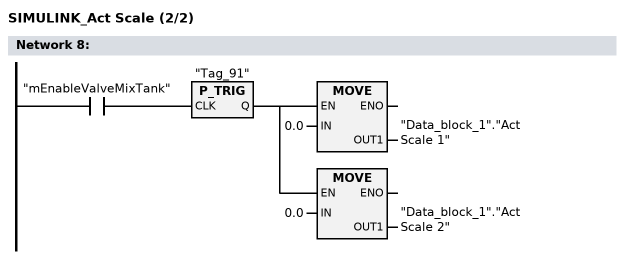
   RUNG wire#powerrail
      Contact( "mEnableValveMixTank" )
      P_Trig( "Tag_91" )
      wire#w1
      Move(in := 0.0, out1 => "Data_block_1"."Act Scale 1")
   END_RUNG
   RUNG wire#w1
      Move(in := 0.0, out1 => "Data_block_1"."Act Scale 2")
   END_RUNG
   // the same network as SCL:
   #_w1 := "mEnableValveMixTank" AND NOT "Tag_91";   // rising edge
   "Tag_91" := "mEnableValveMixTank";
   IF #_w1 THEN
       "Data_block_1"."Act Scale 1" := 0.0;
       "Data_block_1"."Act Scale 2" := 0.0;
   END_IF;
END_REGION
END_FUNCTION

FUNCTION "Xilo_Rice" : Void   // FC4, LAD
{ S7_Optimized_Access := 'TRUE' }
VERSION : 0.1
   VAR_TEMP   // added for the SCL form of the ladder/FBD networks
      _w1 : Bool;
      _w2 : Bool;
      _w3 : Bool;
   END_VAR
BEGIN

REGION Network 1
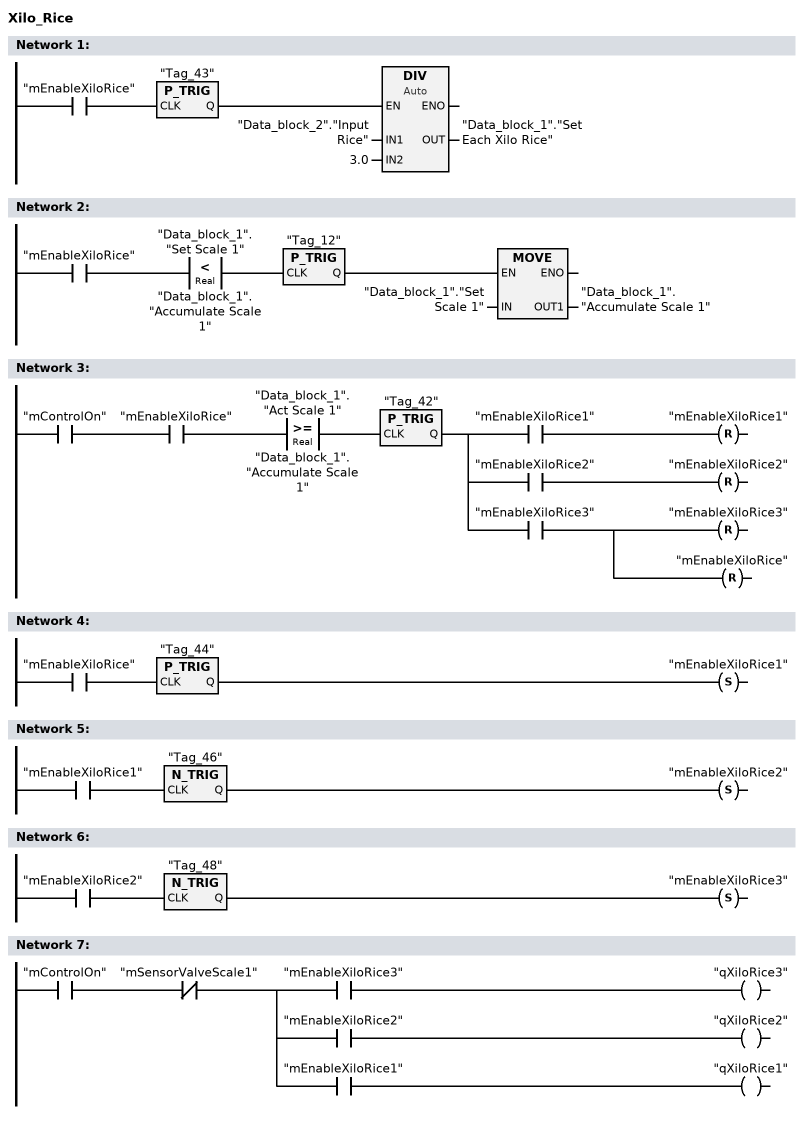
   RUNG wire#powerrail
      Contact( "mEnableXiloRice" )
      P_Trig( "Tag_43" )
      Div(in1 := "Data_block_2"."Input Rice", in2 := 3.0, out => "Data_block_1"."Set Each Xilo Rice")
   END_RUNG
   // the same network as SCL:
   #_w1 := "mEnableXiloRice" AND NOT "Tag_43";   // rising edge
   "Tag_43" := "mEnableXiloRice";
   IF #_w1 THEN "Data_block_1"."Set Each Xilo Rice" := "Data_block_2"."Input Rice" / 3.0; END_IF;
END_REGION

REGION Network 2
   RUNG wire#powerrail
      Contact( "mEnableXiloRice" )
      { S7_Templates := "SrcType := Real" } LT_Contact(in1 := "Data_block_1"."Set Scale 1", in2 := "Data_block_1"."Accumulate Scale 1")
      P_Trig( "Tag_12" )
      Move(in := "Data_block_1"."Set Scale 1", out1 => "Data_block_1"."Accumulate Scale 1")
   END_RUNG
   // the same network as SCL:
   #_w1 := "mEnableXiloRice" AND ("Data_block_1"."Set Scale 1" < "Data_block_1"."Accumulate Scale 1");
   #_w2 := #_w1 AND NOT "Tag_12";   // rising edge
   "Tag_12" := #_w1;
   IF #_w2 THEN "Data_block_1"."Accumulate Scale 1" := "Data_block_1"."Set Scale 1"; END_IF;
END_REGION

REGION Network 3
   RUNG wire#powerrail
      Contact( "mControlOn" )
      Contact( "mEnableXiloRice" )
      { S7_Templates := "SrcType := Real" } GE_Contact(in1 := "Data_block_1"."Act Scale 1", in2 := "Data_block_1"."Accumulate Scale 1")
      P_Trig( "Tag_42" )
      wire#w1
      Contact( "mEnableXiloRice1" )
      R_Coil( "mEnableXiloRice1" )
   END_RUNG
   RUNG wire#w1
      Contact( "mEnableXiloRice2" )
      R_Coil( "mEnableXiloRice2" )
   END_RUNG
   RUNG wire#w1
      Contact( "mEnableXiloRice3" )
      wire#w2
      R_Coil( "mEnableXiloRice3" )
   END_RUNG
   RUNG wire#w2
      R_Coil( "mEnableXiloRice" )
   END_RUNG
   // the same network as SCL:
   #_w1 := "mControlOn" AND "mEnableXiloRice" AND ("Data_block_1"."Act Scale 1" >= "Data_block_1"."Accumulate Scale 1");
   #_w2 := #_w1 AND NOT "Tag_42";   // rising edge
   "Tag_42" := #_w1;
   IF #_w2 AND "mEnableXiloRice1" THEN "mEnableXiloRice1" := FALSE; END_IF;
   IF #_w2 AND "mEnableXiloRice2" THEN "mEnableXiloRice2" := FALSE; END_IF;
   #_w3 := #_w2 AND "mEnableXiloRice3";
   IF #_w3 THEN
       "mEnableXiloRice3" := FALSE;
       "mEnableXiloRice" := FALSE;
   END_IF;
END_REGION

REGION Network 4
   RUNG wire#powerrail
      Contact( "mEnableXiloRice" )
      P_Trig( "Tag_44" )
      S_Coil( "mEnableXiloRice1" )
   END_RUNG
   // the same network as SCL:
   #_w1 := "mEnableXiloRice" AND NOT "Tag_44";   // rising edge
   "Tag_44" := "mEnableXiloRice";
   IF #_w1 THEN "mEnableXiloRice1" := TRUE; END_IF;
END_REGION

REGION Network 5
   RUNG wire#powerrail
      Contact( "mEnableXiloRice1" )
      N_Trig( "Tag_46" )
      S_Coil( "mEnableXiloRice2" )
   END_RUNG
   // the same network as SCL:
   #_w1 := NOT "mEnableXiloRice1" AND "Tag_46";   // falling edge
   "Tag_46" := "mEnableXiloRice1";
   IF #_w1 THEN "mEnableXiloRice2" := TRUE; END_IF;
END_REGION

REGION Network 6
   RUNG wire#powerrail
      Contact( "mEnableXiloRice2" )
      N_Trig( "Tag_48" )
      S_Coil( "mEnableXiloRice3" )
   END_RUNG
   // the same network as SCL:
   #_w1 := NOT "mEnableXiloRice2" AND "Tag_48";   // falling edge
   "Tag_48" := "mEnableXiloRice2";
   IF #_w1 THEN "mEnableXiloRice3" := TRUE; END_IF;
END_REGION

REGION Network 7
   RUNG wire#powerrail
      Contact( "mControlOn" )
      I_Contact( "mSensorValveScale1" )
      wire#w1
      Contact( "mEnableXiloRice3" )
      Coil( "qXiloRice3" )
   END_RUNG
   RUNG wire#w1
      Contact( "mEnableXiloRice2" )
      Coil( "qXiloRice2" )
   END_RUNG
   RUNG wire#w1
      Contact( "mEnableXiloRice1" )
      Coil( "qXiloRice1" )
   END_RUNG
   // the same network as SCL:
   #_w1 := "mControlOn" AND NOT "mSensorValveScale1";
   "qXiloRice3" := #_w1 AND "mEnableXiloRice3";
   "qXiloRice2" := #_w1 AND "mEnableXiloRice2";
   "qXiloRice1" := #_w1 AND "mEnableXiloRice1";
END_REGION
END_FUNCTION

FUNCTION "Control_Inverter" : Void   // FC5, LAD
{ S7_Optimized_Access := 'TRUE' }
VERSION : 0.1
BEGIN

REGION Network 1
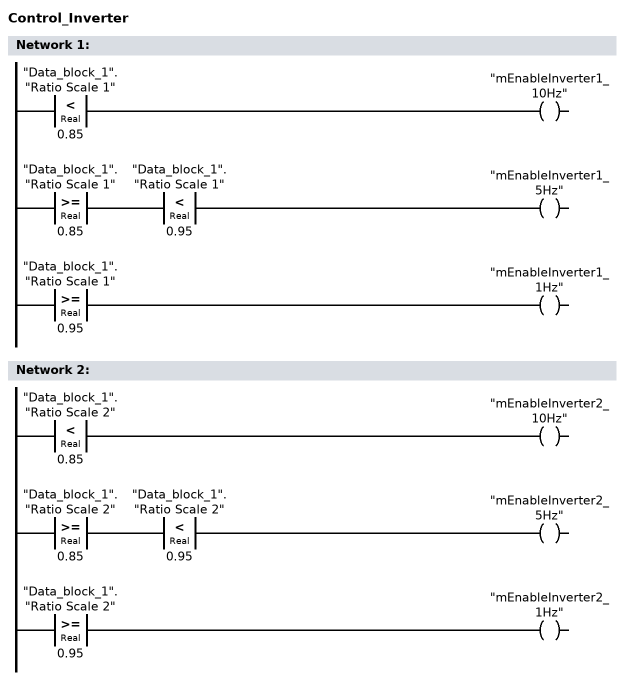
   RUNG wire#powerrail
      { S7_Templates := "SrcType := Real" } LT_Contact(in1 := "Data_block_1"."Ratio Scale 1", in2 := 0.85)
      Coil( "mEnableInverter1_10Hz" )
   END_RUNG
   RUNG wire#powerrail
      { S7_Templates := "SrcType := Real" } GE_Contact(in1 := "Data_block_1"."Ratio Scale 1", in2 := 0.85)
      { S7_Templates := "SrcType := Real" } LT_Contact(in1 := "Data_block_1"."Ratio Scale 1", in2 := 0.95)
      Coil( "mEnableInverter1_5Hz" )
   END_RUNG
   RUNG wire#powerrail
      { S7_Templates := "SrcType := Real" } GE_Contact(in1 := "Data_block_1"."Ratio Scale 1", in2 := 0.95)
      Coil( "mEnableInverter1_1Hz" )
   END_RUNG
   // the same network as SCL:
   "mEnableInverter1_10Hz" := "Data_block_1"."Ratio Scale 1" < 0.85;
   "mEnableInverter1_5Hz" := ("Data_block_1"."Ratio Scale 1" >= 0.85) AND ("Data_block_1"."Ratio Scale 1" < 0.95);
   "mEnableInverter1_1Hz" := "Data_block_1"."Ratio Scale 1" >= 0.95;
END_REGION

REGION Network 2
   RUNG wire#powerrail
      { S7_Templates := "SrcType := Real" } LT_Contact(in1 := "Data_block_1"."Ratio Scale 2", in2 := 0.85)
      Coil( "mEnableInverter2_10Hz" )
   END_RUNG
   RUNG wire#powerrail
      { S7_Templates := "SrcType := Real" } GE_Contact(in1 := "Data_block_1"."Ratio Scale 2", in2 := 0.85)
      { S7_Templates := "SrcType := Real" } LT_Contact(in1 := "Data_block_1"."Ratio Scale 2", in2 := 0.95)
      Coil( "mEnableInverter2_5Hz" )
   END_RUNG
   RUNG wire#powerrail
      { S7_Templates := "SrcType := Real" } GE_Contact(in1 := "Data_block_1"."Ratio Scale 2", in2 := 0.95)
      Coil( "mEnableInverter2_1Hz" )
   END_RUNG
   // the same network as SCL:
   "mEnableInverter2_10Hz" := "Data_block_1"."Ratio Scale 2" < 0.85;
   "mEnableInverter2_5Hz" := ("Data_block_1"."Ratio Scale 2" >= 0.85) AND ("Data_block_1"."Ratio Scale 2" < 0.95);
   "mEnableInverter2_1Hz" := "Data_block_1"."Ratio Scale 2" >= 0.95;
END_REGION
END_FUNCTION

FUNCTION "Xilo_Corn" : Void   // FC6, LAD
{ S7_Optimized_Access := 'TRUE' }
VERSION : 0.1
   VAR_TEMP   // added for the SCL form of the ladder/FBD networks
      _w1 : Bool;
      _w2 : Bool;
      _w3 : Bool;
   END_VAR
BEGIN

REGION Network 1
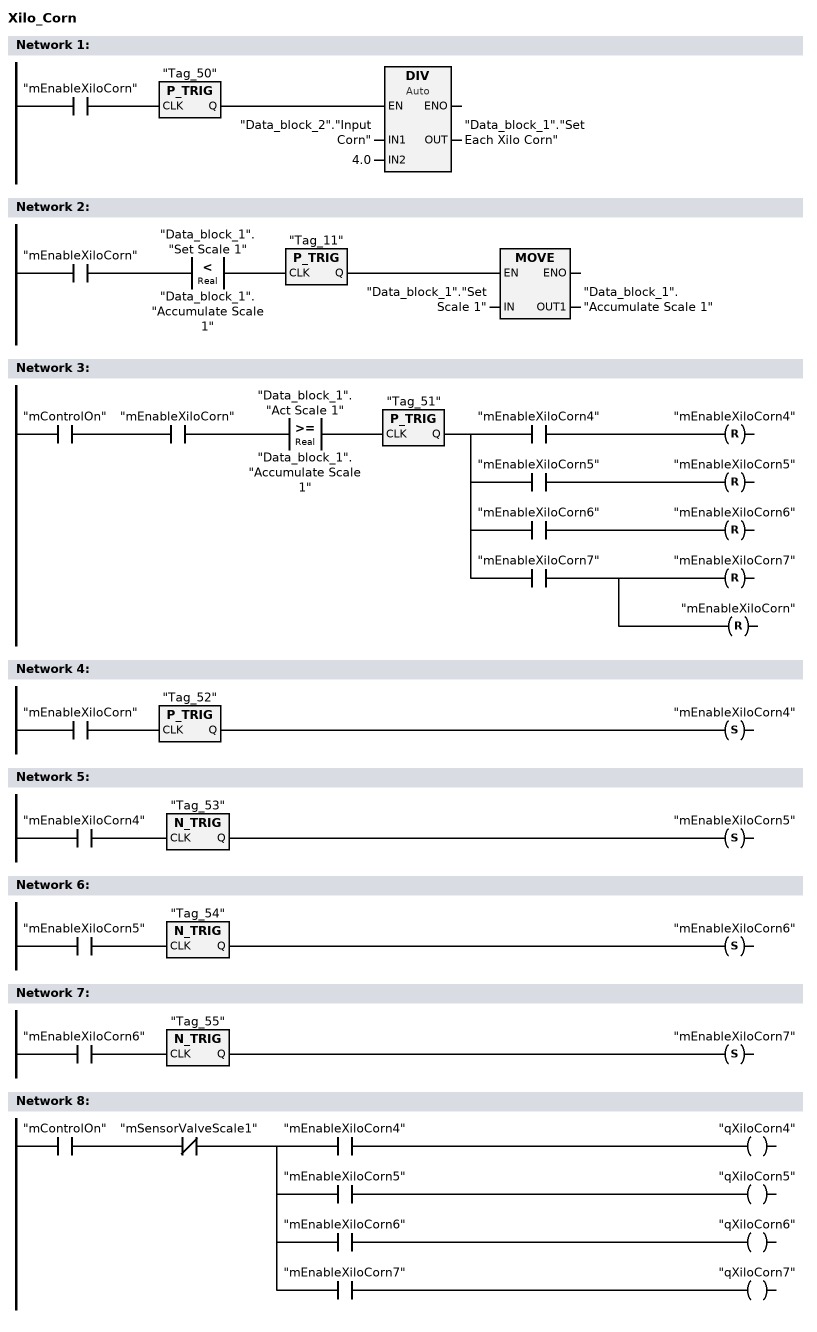
   RUNG wire#powerrail
      Contact( "mEnableXiloCorn" )
      P_Trig( "Tag_50" )
      Div(in1 := "Data_block_2"."Input Corn", in2 := 4.0, out => "Data_block_1"."Set Each Xilo Corn")
   END_RUNG
   // the same network as SCL:
   #_w1 := "mEnableXiloCorn" AND NOT "Tag_50";   // rising edge
   "Tag_50" := "mEnableXiloCorn";
   IF #_w1 THEN "Data_block_1"."Set Each Xilo Corn" := "Data_block_2"."Input Corn" / 4.0; END_IF;
END_REGION

REGION Network 2
   RUNG wire#powerrail
      Contact( "mEnableXiloCorn" )
      { S7_Templates := "SrcType := Real" } LT_Contact(in1 := "Data_block_1"."Set Scale 1", in2 := "Data_block_1"."Accumulate Scale 1")
      P_Trig( "Tag_11" )
      Move(in := "Data_block_1"."Set Scale 1", out1 => "Data_block_1"."Accumulate Scale 1")
   END_RUNG
   // the same network as SCL:
   #_w1 := "mEnableXiloCorn" AND ("Data_block_1"."Set Scale 1" < "Data_block_1"."Accumulate Scale 1");
   #_w2 := #_w1 AND NOT "Tag_11";   // rising edge
   "Tag_11" := #_w1;
   IF #_w2 THEN "Data_block_1"."Accumulate Scale 1" := "Data_block_1"."Set Scale 1"; END_IF;
END_REGION

REGION Network 3
   RUNG wire#powerrail
      Contact( "mControlOn" )
      Contact( "mEnableXiloCorn" )
      { S7_Templates := "SrcType := Real" } GE_Contact(in1 := "Data_block_1"."Act Scale 1", in2 := "Data_block_1"."Accumulate Scale 1")
      P_Trig( "Tag_51" )
      wire#w1
      Contact( "mEnableXiloCorn4" )
      R_Coil( "mEnableXiloCorn4" )
   END_RUNG
   RUNG wire#w1
      Contact( "mEnableXiloCorn5" )
      R_Coil( "mEnableXiloCorn5" )
   END_RUNG
   RUNG wire#w1
      Contact( "mEnableXiloCorn6" )
      R_Coil( "mEnableXiloCorn6" )
   END_RUNG
   RUNG wire#w1
      Contact( "mEnableXiloCorn7" )
      wire#w2
      R_Coil( "mEnableXiloCorn7" )
   END_RUNG
   RUNG wire#w2
      R_Coil( "mEnableXiloCorn" )
   END_RUNG
   // the same network as SCL:
   #_w1 := "mControlOn" AND "mEnableXiloCorn" AND ("Data_block_1"."Act Scale 1" >= "Data_block_1"."Accumulate Scale 1");
   #_w2 := #_w1 AND NOT "Tag_51";   // rising edge
   "Tag_51" := #_w1;
   IF #_w2 AND "mEnableXiloCorn4" THEN "mEnableXiloCorn4" := FALSE; END_IF;
   IF #_w2 AND "mEnableXiloCorn5" THEN "mEnableXiloCorn5" := FALSE; END_IF;
   IF #_w2 AND "mEnableXiloCorn6" THEN "mEnableXiloCorn6" := FALSE; END_IF;
   #_w3 := #_w2 AND "mEnableXiloCorn7";
   IF #_w3 THEN
       "mEnableXiloCorn7" := FALSE;
       "mEnableXiloCorn" := FALSE;
   END_IF;
END_REGION

REGION Network 4
   RUNG wire#powerrail
      Contact( "mEnableXiloCorn" )
      P_Trig( "Tag_52" )
      S_Coil( "mEnableXiloCorn4" )
   END_RUNG
   // the same network as SCL:
   #_w1 := "mEnableXiloCorn" AND NOT "Tag_52";   // rising edge
   "Tag_52" := "mEnableXiloCorn";
   IF #_w1 THEN "mEnableXiloCorn4" := TRUE; END_IF;
END_REGION

REGION Network 5
   RUNG wire#powerrail
      Contact( "mEnableXiloCorn4" )
      N_Trig( "Tag_53" )
      S_Coil( "mEnableXiloCorn5" )
   END_RUNG
   // the same network as SCL:
   #_w1 := NOT "mEnableXiloCorn4" AND "Tag_53";   // falling edge
   "Tag_53" := "mEnableXiloCorn4";
   IF #_w1 THEN "mEnableXiloCorn5" := TRUE; END_IF;
END_REGION

REGION Network 6
   RUNG wire#powerrail
      Contact( "mEnableXiloCorn5" )
      N_Trig( "Tag_54" )
      S_Coil( "mEnableXiloCorn6" )
   END_RUNG
   // the same network as SCL:
   #_w1 := NOT "mEnableXiloCorn5" AND "Tag_54";   // falling edge
   "Tag_54" := "mEnableXiloCorn5";
   IF #_w1 THEN "mEnableXiloCorn6" := TRUE; END_IF;
END_REGION

REGION Network 7
   RUNG wire#powerrail
      Contact( "mEnableXiloCorn6" )
      N_Trig( "Tag_55" )
      S_Coil( "mEnableXiloCorn7" )
   END_RUNG
   // the same network as SCL:
   #_w1 := NOT "mEnableXiloCorn6" AND "Tag_55";   // falling edge
   "Tag_55" := "mEnableXiloCorn6";
   IF #_w1 THEN "mEnableXiloCorn7" := TRUE; END_IF;
END_REGION

REGION Network 8
   RUNG wire#powerrail
      Contact( "mControlOn" )
      I_Contact( "mSensorValveScale1" )
      wire#w1
      Contact( "mEnableXiloCorn4" )
      Coil( "qXiloCorn4" )
   END_RUNG
   RUNG wire#w1
      Contact( "mEnableXiloCorn5" )
      Coil( "qXiloCorn5" )
   END_RUNG
   RUNG wire#w1
      Contact( "mEnableXiloCorn6" )
      Coil( "qXiloCorn6" )
   END_RUNG
   RUNG wire#w1
      Contact( "mEnableXiloCorn7" )
      Coil( "qXiloCorn7" )
   END_RUNG
   // the same network as SCL:
   #_w1 := "mControlOn" AND NOT "mSensorValveScale1";
   "qXiloCorn4" := #_w1 AND "mEnableXiloCorn4";
   "qXiloCorn5" := #_w1 AND "mEnableXiloCorn5";
   "qXiloCorn6" := #_w1 AND "mEnableXiloCorn6";
   "qXiloCorn7" := #_w1 AND "mEnableXiloCorn7";
END_REGION
END_FUNCTION

FUNCTION "Xilo_Cassava" : Void   // FC7, LAD
{ S7_Optimized_Access := 'TRUE' }
VERSION : 0.1
   VAR_TEMP   // added for the SCL form of the ladder/FBD networks
      _w1 : Bool;
      _w2 : Bool;
      _w3 : Bool;
   END_VAR
BEGIN

REGION Network 1
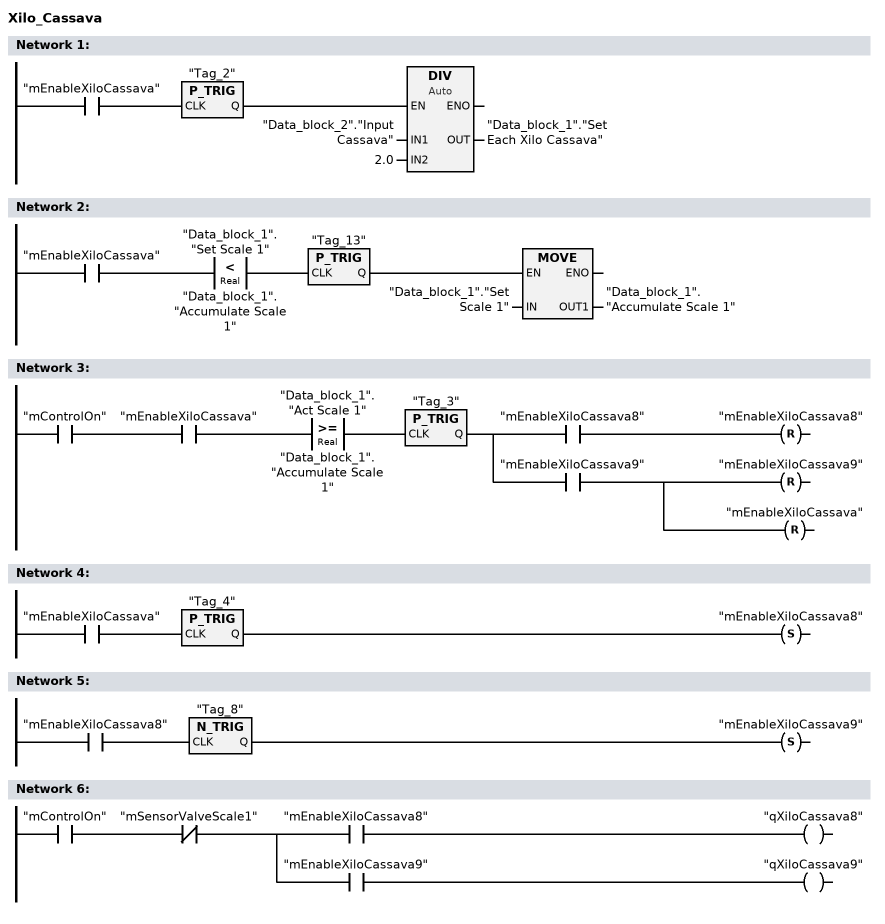
   RUNG wire#powerrail
      Contact( "mEnableXiloCassava" )
      P_Trig( "Tag_2" )
      Div(in1 := "Data_block_2"."Input Cassava", in2 := 2.0, out => "Data_block_1"."Set Each Xilo Cassava")
   END_RUNG
   // the same network as SCL:
   #_w1 := "mEnableXiloCassava" AND NOT "Tag_2";   // rising edge
   "Tag_2" := "mEnableXiloCassava";
   IF #_w1 THEN "Data_block_1"."Set Each Xilo Cassava" := "Data_block_2"."Input Cassava" / 2.0; END_IF;
END_REGION

REGION Network 2
   RUNG wire#powerrail
      Contact( "mEnableXiloCassava" )
      { S7_Templates := "SrcType := Real" } LT_Contact(in1 := "Data_block_1"."Set Scale 1", in2 := "Data_block_1"."Accumulate Scale 1")
      P_Trig( "Tag_13" )
      Move(in := "Data_block_1"."Set Scale 1", out1 => "Data_block_1"."Accumulate Scale 1")
   END_RUNG
   // the same network as SCL:
   #_w1 := "mEnableXiloCassava" AND ("Data_block_1"."Set Scale 1" < "Data_block_1"."Accumulate Scale 1");
   #_w2 := #_w1 AND NOT "Tag_13";   // rising edge
   "Tag_13" := #_w1;
   IF #_w2 THEN "Data_block_1"."Accumulate Scale 1" := "Data_block_1"."Set Scale 1"; END_IF;
END_REGION

REGION Network 3
   RUNG wire#powerrail
      Contact( "mControlOn" )
      Contact( "mEnableXiloCassava" )
      { S7_Templates := "SrcType := Real" } GE_Contact(in1 := "Data_block_1"."Act Scale 1", in2 := "Data_block_1"."Accumulate Scale 1")
      P_Trig( "Tag_3" )
      wire#w1
      Contact( "mEnableXiloCassava8" )
      R_Coil( "mEnableXiloCassava8" )
   END_RUNG
   RUNG wire#w1
      Contact( "mEnableXiloCassava9" )
      wire#w2
      R_Coil( "mEnableXiloCassava9" )
   END_RUNG
   RUNG wire#w2
      R_Coil( "mEnableXiloCassava" )
   END_RUNG
   // the same network as SCL:
   #_w1 := "mControlOn" AND "mEnableXiloCassava" AND ("Data_block_1"."Act Scale 1" >= "Data_block_1"."Accumulate Scale 1");
   #_w2 := #_w1 AND NOT "Tag_3";   // rising edge
   "Tag_3" := #_w1;
   IF #_w2 AND "mEnableXiloCassava8" THEN "mEnableXiloCassava8" := FALSE; END_IF;
   #_w3 := #_w2 AND "mEnableXiloCassava9";
   IF #_w3 THEN
       "mEnableXiloCassava9" := FALSE;
       "mEnableXiloCassava" := FALSE;
   END_IF;
END_REGION

REGION Network 4
   RUNG wire#powerrail
      Contact( "mEnableXiloCassava" )
      P_Trig( "Tag_4" )
      S_Coil( "mEnableXiloCassava8" )
   END_RUNG
   // the same network as SCL:
   #_w1 := "mEnableXiloCassava" AND NOT "Tag_4";   // rising edge
   "Tag_4" := "mEnableXiloCassava";
   IF #_w1 THEN "mEnableXiloCassava8" := TRUE; END_IF;
END_REGION

REGION Network 5
   RUNG wire#powerrail
      Contact( "mEnableXiloCassava8" )
      N_Trig( "Tag_8" )
      S_Coil( "mEnableXiloCassava9" )
   END_RUNG
   // the same network as SCL:
   #_w1 := NOT "mEnableXiloCassava8" AND "Tag_8";   // falling edge
   "Tag_8" := "mEnableXiloCassava8";
   IF #_w1 THEN "mEnableXiloCassava9" := TRUE; END_IF;
END_REGION

REGION Network 6
   RUNG wire#powerrail
      Contact( "mControlOn" )
      I_Contact( "mSensorValveScale1" )
      wire#w1
      Contact( "mEnableXiloCassava8" )
      Coil( "qXiloCassava8" )
   END_RUNG
   RUNG wire#w1
      Contact( "mEnableXiloCassava9" )
      Coil( "qXiloCassava9" )
   END_RUNG
   // the same network as SCL:
   #_w1 := "mControlOn" AND NOT "mSensorValveScale1";
   "qXiloCassava8" := #_w1 AND "mEnableXiloCassava8";
   "qXiloCassava9" := #_w1 AND "mEnableXiloCassava9";
END_REGION
END_FUNCTION

FUNCTION "Select_Xilo_Scale2" : Void   // FC8, LAD
{ S7_Optimized_Access := 'TRUE' }
VERSION : 0.1
   VAR_TEMP   // added for the SCL form of the ladder/FBD networks
      _w1 : Bool;
      _w2 : Bool;
   END_VAR
BEGIN

REGION Network 1
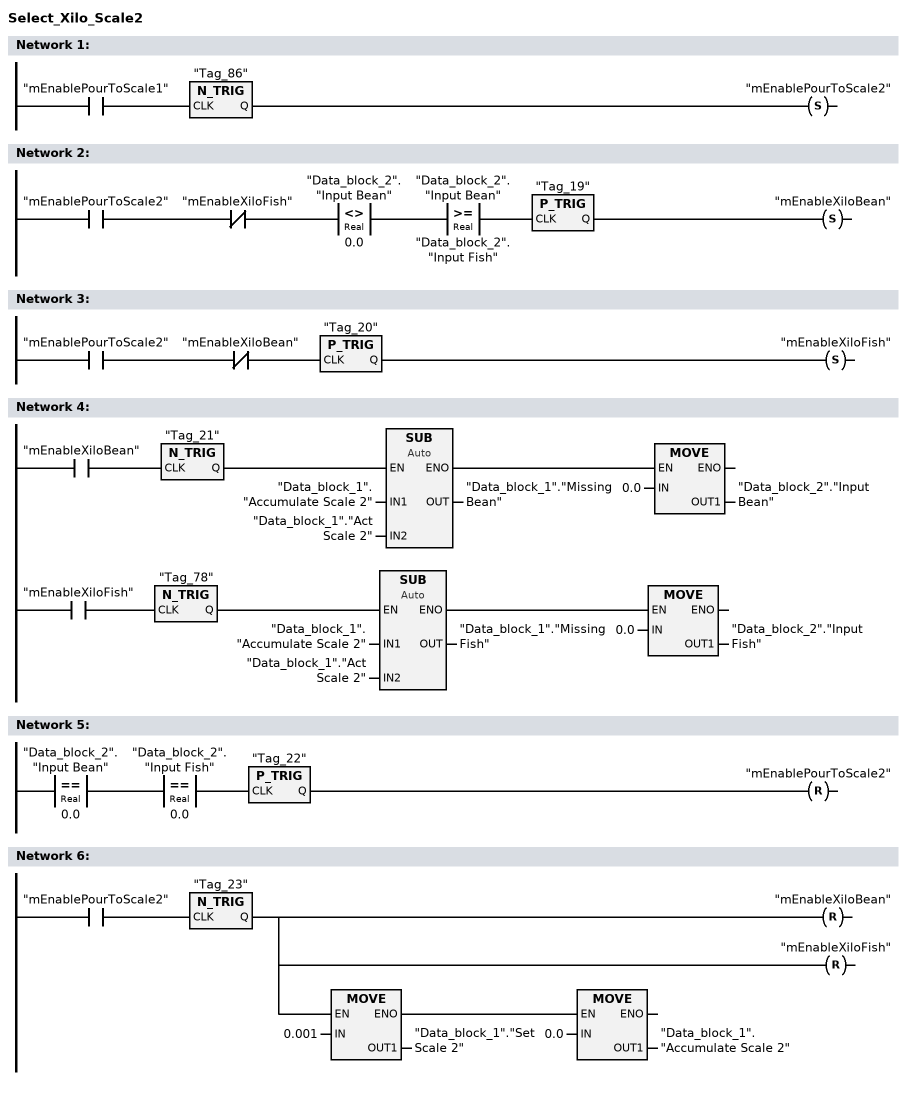
   RUNG wire#powerrail
      Contact( "mEnablePourToScale1" )
      N_Trig( "Tag_86" )
      S_Coil( "mEnablePourToScale2" )
   END_RUNG
   // the same network as SCL:
   #_w1 := NOT "mEnablePourToScale1" AND "Tag_86";   // falling edge
   "Tag_86" := "mEnablePourToScale1";
   IF #_w1 THEN "mEnablePourToScale2" := TRUE; END_IF;
END_REGION

REGION Network 2
   RUNG wire#powerrail
      Contact( "mEnablePourToScale2" )
      I_Contact( "mEnableXiloFish" )
      { S7_Templates := "SrcType := Real" } NE_Contact(in1 := "Data_block_2"."Input Bean", in2 := 0.0)
      { S7_Templates := "SrcType := Real" } GE_Contact(in1 := "Data_block_2"."Input Bean", in2 := "Data_block_2"."Input Fish")
      P_Trig( "Tag_19" )
      S_Coil( "mEnableXiloBean" )
   END_RUNG
   // the same network as SCL:
   #_w1 := "mEnablePourToScale2" AND NOT "mEnableXiloFish" AND ("Data_block_2"."Input Bean" <> 0.0) AND ("Data_block_2"."Input Bean" >= "Data_block_2"."Input Fish");
   #_w2 := #_w1 AND NOT "Tag_19";   // rising edge
   "Tag_19" := #_w1;
   IF #_w2 THEN "mEnableXiloBean" := TRUE; END_IF;
END_REGION

REGION Network 3
   RUNG wire#powerrail
      Contact( "mEnablePourToScale2" )
      I_Contact( "mEnableXiloBean" )
      P_Trig( "Tag_20" )
      S_Coil( "mEnableXiloFish" )
   END_RUNG
   // the same network as SCL:
   #_w1 := "mEnablePourToScale2" AND NOT "mEnableXiloBean";
   #_w2 := #_w1 AND NOT "Tag_20";   // rising edge
   "Tag_20" := #_w1;
   IF #_w2 THEN "mEnableXiloFish" := TRUE; END_IF;
END_REGION

REGION Network 4
   RUNG wire#powerrail
      Contact( "mEnableXiloBean" )
      N_Trig( "Tag_21" )
      Sub(in1 := "Data_block_1"."Accumulate Scale 2", in2 := "Data_block_1"."Act Scale 2", out => "Data_block_1"."Missing Bean")
      Move(in := 0.0, out1 => "Data_block_2"."Input Bean")
   END_RUNG
   RUNG wire#powerrail
      Contact( "mEnableXiloFish" )
      N_Trig( "Tag_78" )
      Sub(in1 := "Data_block_1"."Accumulate Scale 2", in2 := "Data_block_1"."Act Scale 2", out => "Data_block_1"."Missing Fish")
      Move(in := 0.0, out1 => "Data_block_2"."Input Fish")
   END_RUNG
   // the same network as SCL:
   #_w1 := NOT "mEnableXiloBean" AND "Tag_21";   // falling edge
   "Tag_21" := "mEnableXiloBean";
   IF #_w1 THEN
       "Data_block_1"."Missing Bean" := "Data_block_1"."Accumulate Scale 2" - "Data_block_1"."Act Scale 2";
       "Data_block_2"."Input Bean" := 0.0;
   END_IF;
   #_w2 := NOT "mEnableXiloFish" AND "Tag_78";   // falling edge
   "Tag_78" := "mEnableXiloFish";
   IF #_w2 THEN
       "Data_block_1"."Missing Fish" := "Data_block_1"."Accumulate Scale 2" - "Data_block_1"."Act Scale 2";
       "Data_block_2"."Input Fish" := 0.0;
   END_IF;
END_REGION

REGION Network 5
   RUNG wire#powerrail
      { S7_Templates := "SrcType := Real" } EQ_Contact(in1 := "Data_block_2"."Input Bean", in2 := 0.0)
      { S7_Templates := "SrcType := Real" } EQ_Contact(in1 := "Data_block_2"."Input Fish", in2 := 0.0)
      P_Trig( "Tag_22" )
      R_Coil( "mEnablePourToScale2" )
   END_RUNG
   // the same network as SCL:
   #_w1 := ("Data_block_2"."Input Bean" = 0.0) AND ("Data_block_2"."Input Fish" = 0.0);
   #_w2 := #_w1 AND NOT "Tag_22";   // rising edge
   "Tag_22" := #_w1;
   IF #_w2 THEN "mEnablePourToScale2" := FALSE; END_IF;
END_REGION

REGION Network 6
   RUNG wire#powerrail
      Contact( "mEnablePourToScale2" )
      N_Trig( "Tag_23" )
      wire#w1
      R_Coil( "mEnableXiloBean" )
   END_RUNG
   RUNG wire#w1
      R_Coil( "mEnableXiloFish" )
   END_RUNG
   RUNG wire#w1
      Move(in := 0.001, out1 => "Data_block_1"."Set Scale 2")
      Move(in := 0.0, out1 => "Data_block_1"."Accumulate Scale 2")
   END_RUNG
   // the same network as SCL:
   #_w1 := NOT "mEnablePourToScale2" AND "Tag_23";   // falling edge
   "Tag_23" := "mEnablePourToScale2";
   IF #_w1 THEN
       "mEnableXiloBean" := FALSE;
       "mEnableXiloFish" := FALSE;
       "Data_block_1"."Set Scale 2" := 0.001;
       "Data_block_1"."Accumulate Scale 2" := 0.0;
   END_IF;
END_REGION
END_FUNCTION

FUNCTION "Xilo_Bean" : Void   // FC9, LAD
{ S7_Optimized_Access := 'TRUE' }
VERSION : 0.1
   VAR_TEMP   // added for the SCL form of the ladder/FBD networks
      _w1 : Bool;
      _w2 : Bool;
      _w3 : Bool;
   END_VAR
BEGIN

REGION Network 1
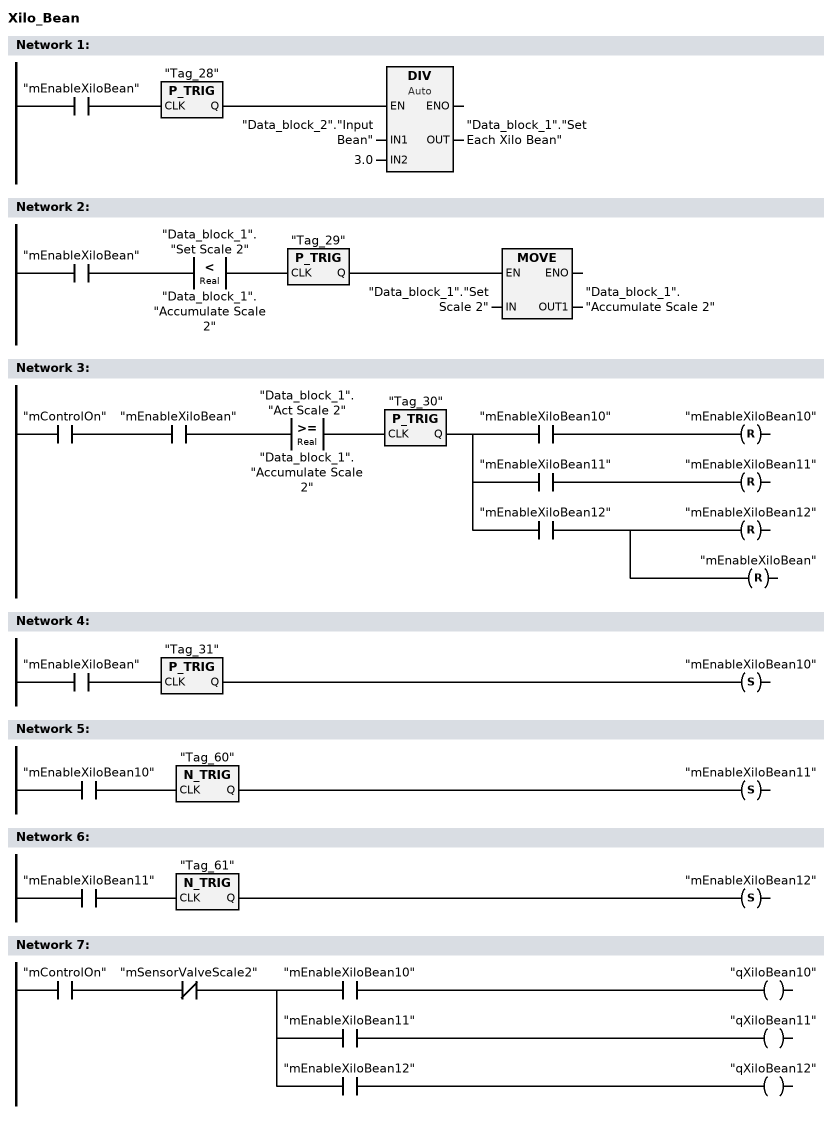
   RUNG wire#powerrail
      Contact( "mEnableXiloBean" )
      P_Trig( "Tag_28" )
      Div(in1 := "Data_block_2"."Input Bean", in2 := 3.0, out => "Data_block_1"."Set Each Xilo Bean")
   END_RUNG
   // the same network as SCL:
   #_w1 := "mEnableXiloBean" AND NOT "Tag_28";   // rising edge
   "Tag_28" := "mEnableXiloBean";
   IF #_w1 THEN "Data_block_1"."Set Each Xilo Bean" := "Data_block_2"."Input Bean" / 3.0; END_IF;
END_REGION

REGION Network 2
   RUNG wire#powerrail
      Contact( "mEnableXiloBean" )
      { S7_Templates := "SrcType := Real" } LT_Contact(in1 := "Data_block_1"."Set Scale 2", in2 := "Data_block_1"."Accumulate Scale 2")
      P_Trig( "Tag_29" )
      Move(in := "Data_block_1"."Set Scale 2", out1 => "Data_block_1"."Accumulate Scale 2")
   END_RUNG
   // the same network as SCL:
   #_w1 := "mEnableXiloBean" AND ("Data_block_1"."Set Scale 2" < "Data_block_1"."Accumulate Scale 2");
   #_w2 := #_w1 AND NOT "Tag_29";   // rising edge
   "Tag_29" := #_w1;
   IF #_w2 THEN "Data_block_1"."Accumulate Scale 2" := "Data_block_1"."Set Scale 2"; END_IF;
END_REGION

REGION Network 3
   RUNG wire#powerrail
      Contact( "mControlOn" )
      Contact( "mEnableXiloBean" )
      { S7_Templates := "SrcType := Real" } GE_Contact(in1 := "Data_block_1"."Act Scale 2", in2 := "Data_block_1"."Accumulate Scale 2")
      P_Trig( "Tag_30" )
      wire#w1
      Contact( "mEnableXiloBean10" )
      R_Coil( "mEnableXiloBean10" )
   END_RUNG
   RUNG wire#w1
      Contact( "mEnableXiloBean11" )
      R_Coil( "mEnableXiloBean11" )
   END_RUNG
   RUNG wire#w1
      Contact( "mEnableXiloBean12" )
      wire#w2
      R_Coil( "mEnableXiloBean12" )
   END_RUNG
   RUNG wire#w2
      R_Coil( "mEnableXiloBean" )
   END_RUNG
   // the same network as SCL:
   #_w1 := "mControlOn" AND "mEnableXiloBean" AND ("Data_block_1"."Act Scale 2" >= "Data_block_1"."Accumulate Scale 2");
   #_w2 := #_w1 AND NOT "Tag_30";   // rising edge
   "Tag_30" := #_w1;
   IF #_w2 AND "mEnableXiloBean10" THEN "mEnableXiloBean10" := FALSE; END_IF;
   IF #_w2 AND "mEnableXiloBean11" THEN "mEnableXiloBean11" := FALSE; END_IF;
   #_w3 := #_w2 AND "mEnableXiloBean12";
   IF #_w3 THEN
       "mEnableXiloBean12" := FALSE;
       "mEnableXiloBean" := FALSE;
   END_IF;
END_REGION

REGION Network 4
   RUNG wire#powerrail
      Contact( "mEnableXiloBean" )
      P_Trig( "Tag_31" )
      S_Coil( "mEnableXiloBean10" )
   END_RUNG
   // the same network as SCL:
   #_w1 := "mEnableXiloBean" AND NOT "Tag_31";   // rising edge
   "Tag_31" := "mEnableXiloBean";
   IF #_w1 THEN "mEnableXiloBean10" := TRUE; END_IF;
END_REGION

REGION Network 5
   RUNG wire#powerrail
      Contact( "mEnableXiloBean10" )
      N_Trig( "Tag_60" )
      S_Coil( "mEnableXiloBean11" )
   END_RUNG
   // the same network as SCL:
   #_w1 := NOT "mEnableXiloBean10" AND "Tag_60";   // falling edge
   "Tag_60" := "mEnableXiloBean10";
   IF #_w1 THEN "mEnableXiloBean11" := TRUE; END_IF;
END_REGION

REGION Network 6
   RUNG wire#powerrail
      Contact( "mEnableXiloBean11" )
      N_Trig( "Tag_61" )
      S_Coil( "mEnableXiloBean12" )
   END_RUNG
   // the same network as SCL:
   #_w1 := NOT "mEnableXiloBean11" AND "Tag_61";   // falling edge
   "Tag_61" := "mEnableXiloBean11";
   IF #_w1 THEN "mEnableXiloBean12" := TRUE; END_IF;
END_REGION

REGION Network 7
   RUNG wire#powerrail
      Contact( "mControlOn" )
      I_Contact( "mSensorValveScale2" )
      wire#w1
      Contact( "mEnableXiloBean10" )
      Coil( "qXiloBean10" )
   END_RUNG
   RUNG wire#w1
      Contact( "mEnableXiloBean11" )
      Coil( "qXiloBean11" )
   END_RUNG
   RUNG wire#w1
      Contact( "mEnableXiloBean12" )
      Coil( "qXiloBean12" )
   END_RUNG
   // the same network as SCL:
   #_w1 := "mControlOn" AND NOT "mSensorValveScale2";
   "qXiloBean10" := #_w1 AND "mEnableXiloBean10";
   "qXiloBean11" := #_w1 AND "mEnableXiloBean11";
   "qXiloBean12" := #_w1 AND "mEnableXiloBean12";
END_REGION
END_FUNCTION

FUNCTION "Sensor_Xilo" : Void   // FC10, LAD
{ S7_Optimized_Access := 'TRUE' }
VERSION : 0.1
   VAR_TEMP   // added for the SCL form of the ladder/FBD networks
      _w1 : Bool;
   END_VAR
BEGIN

REGION Network 1
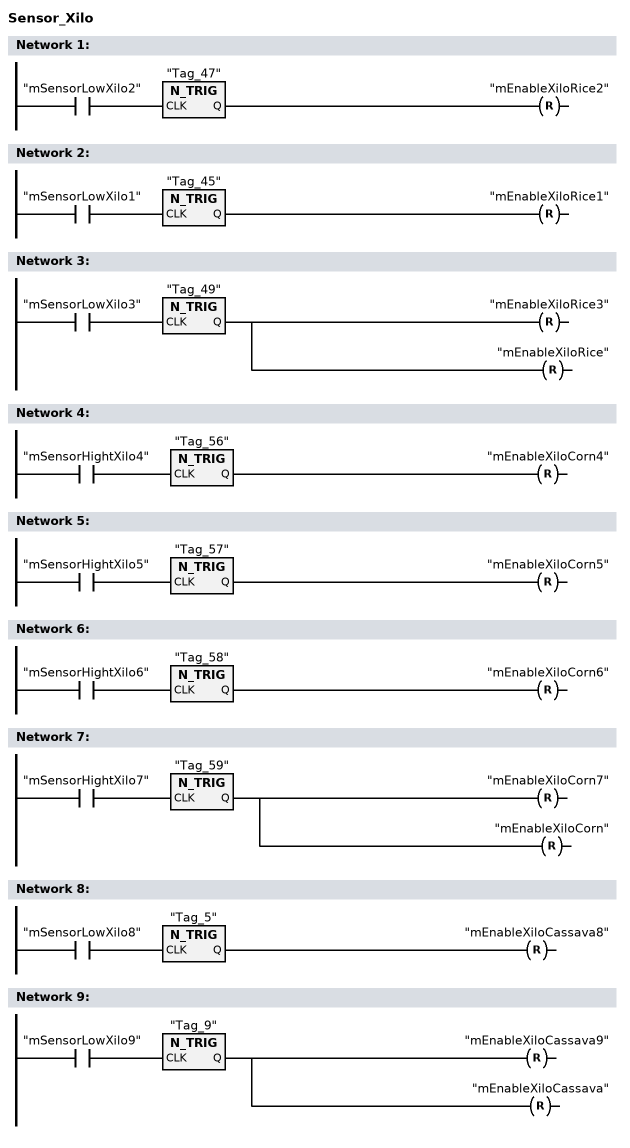
   RUNG wire#powerrail
      Contact( "mSensorLowXilo2" )
      N_Trig( "Tag_47" )
      R_Coil( "mEnableXiloRice2" )
   END_RUNG
   // the same network as SCL:
   #_w1 := NOT "mSensorLowXilo2" AND "Tag_47";   // falling edge
   "Tag_47" := "mSensorLowXilo2";
   IF #_w1 THEN "mEnableXiloRice2" := FALSE; END_IF;
END_REGION

REGION Network 2
   RUNG wire#powerrail
      Contact( "mSensorLowXilo1" )
      N_Trig( "Tag_45" )
      R_Coil( "mEnableXiloRice1" )
   END_RUNG
   // the same network as SCL:
   #_w1 := NOT "mSensorLowXilo1" AND "Tag_45";   // falling edge
   "Tag_45" := "mSensorLowXilo1";
   IF #_w1 THEN "mEnableXiloRice1" := FALSE; END_IF;
END_REGION

REGION Network 3
   RUNG wire#powerrail
      Contact( "mSensorLowXilo3" )
      N_Trig( "Tag_49" )
      wire#w1
      R_Coil( "mEnableXiloRice3" )
   END_RUNG
   RUNG wire#w1
      R_Coil( "mEnableXiloRice" )
   END_RUNG
   // the same network as SCL:
   #_w1 := NOT "mSensorLowXilo3" AND "Tag_49";   // falling edge
   "Tag_49" := "mSensorLowXilo3";
   IF #_w1 THEN
       "mEnableXiloRice3" := FALSE;
       "mEnableXiloRice" := FALSE;
   END_IF;
END_REGION

REGION Network 4
   RUNG wire#powerrail
      Contact( "mSensorHightXilo4" )
      N_Trig( "Tag_56" )
      R_Coil( "mEnableXiloCorn4" )
   END_RUNG
   // the same network as SCL:
   #_w1 := NOT "mSensorHightXilo4" AND "Tag_56";   // falling edge
   "Tag_56" := "mSensorHightXilo4";
   IF #_w1 THEN "mEnableXiloCorn4" := FALSE; END_IF;
END_REGION

REGION Network 5
   RUNG wire#powerrail
      Contact( "mSensorHightXilo5" )
      N_Trig( "Tag_57" )
      R_Coil( "mEnableXiloCorn5" )
   END_RUNG
   // the same network as SCL:
   #_w1 := NOT "mSensorHightXilo5" AND "Tag_57";   // falling edge
   "Tag_57" := "mSensorHightXilo5";
   IF #_w1 THEN "mEnableXiloCorn5" := FALSE; END_IF;
END_REGION

REGION Network 6
   RUNG wire#powerrail
      Contact( "mSensorHightXilo6" )
      N_Trig( "Tag_58" )
      R_Coil( "mEnableXiloCorn6" )
   END_RUNG
   // the same network as SCL:
   #_w1 := NOT "mSensorHightXilo6" AND "Tag_58";   // falling edge
   "Tag_58" := "mSensorHightXilo6";
   IF #_w1 THEN "mEnableXiloCorn6" := FALSE; END_IF;
END_REGION

REGION Network 7
   RUNG wire#powerrail
      Contact( "mSensorHightXilo7" )
      N_Trig( "Tag_59" )
      wire#w1
      R_Coil( "mEnableXiloCorn7" )
   END_RUNG
   RUNG wire#w1
      R_Coil( "mEnableXiloCorn" )
   END_RUNG
   // the same network as SCL:
   #_w1 := NOT "mSensorHightXilo7" AND "Tag_59";   // falling edge
   "Tag_59" := "mSensorHightXilo7";
   IF #_w1 THEN
       "mEnableXiloCorn7" := FALSE;
       "mEnableXiloCorn" := FALSE;
   END_IF;
END_REGION

REGION Network 8
   RUNG wire#powerrail
      Contact( "mSensorLowXilo8" )
      N_Trig( "Tag_5" )
      R_Coil( "mEnableXiloCassava8" )
   END_RUNG
   // the same network as SCL:
   #_w1 := NOT "mSensorLowXilo8" AND "Tag_5";   // falling edge
   "Tag_5" := "mSensorLowXilo8";
   IF #_w1 THEN "mEnableXiloCassava8" := FALSE; END_IF;
END_REGION

REGION Network 9
   RUNG wire#powerrail
      Contact( "mSensorLowXilo9" )
      N_Trig( "Tag_9" )
      wire#w1
      R_Coil( "mEnableXiloCassava9" )
   END_RUNG
   RUNG wire#w1
      R_Coil( "mEnableXiloCassava" )
   END_RUNG
   // the same network as SCL:
   #_w1 := NOT "mSensorLowXilo9" AND "Tag_9";   // falling edge
   "Tag_9" := "mSensorLowXilo9";
   IF #_w1 THEN
       "mEnableXiloCassava9" := FALSE;
       "mEnableXiloCassava" := FALSE;
   END_IF;
END_REGION
END_FUNCTION

FUNCTION "Xilo_Fish" : Void   // FC11, LAD
{ S7_Optimized_Access := 'TRUE' }
VERSION : 0.1
   VAR_TEMP   // added for the SCL form of the ladder/FBD networks
      _w1 : Bool;
      _w2 : Bool;
      _w3 : Bool;
   END_VAR
BEGIN

REGION Network 1
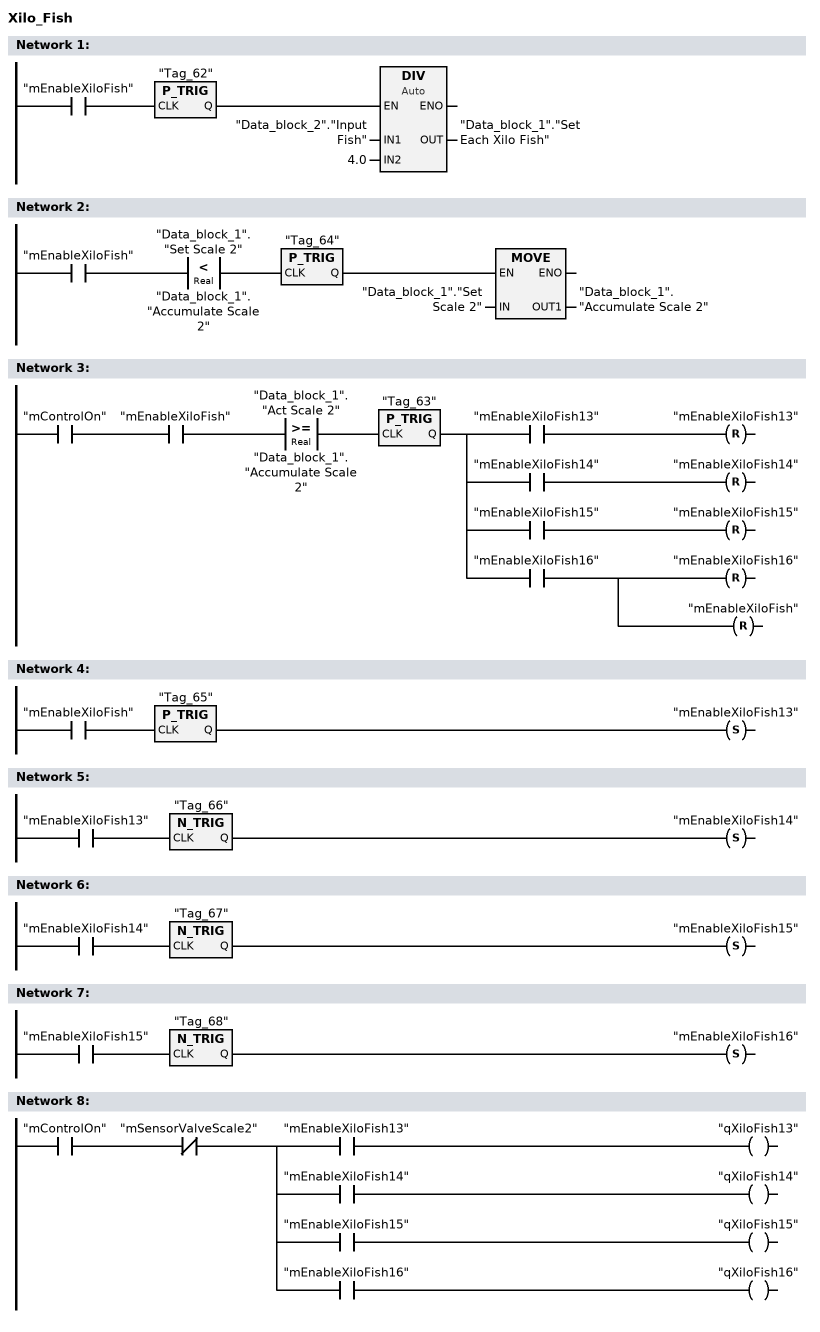
   RUNG wire#powerrail
      Contact( "mEnableXiloFish" )
      P_Trig( "Tag_62" )
      Div(in1 := "Data_block_2"."Input Fish", in2 := 4.0, out => "Data_block_1"."Set Each Xilo Fish")
   END_RUNG
   // the same network as SCL:
   #_w1 := "mEnableXiloFish" AND NOT "Tag_62";   // rising edge
   "Tag_62" := "mEnableXiloFish";
   IF #_w1 THEN "Data_block_1"."Set Each Xilo Fish" := "Data_block_2"."Input Fish" / 4.0; END_IF;
END_REGION

REGION Network 2
   RUNG wire#powerrail
      Contact( "mEnableXiloFish" )
      { S7_Templates := "SrcType := Real" } LT_Contact(in1 := "Data_block_1"."Set Scale 2", in2 := "Data_block_1"."Accumulate Scale 2")
      P_Trig( "Tag_64" )
      Move(in := "Data_block_1"."Set Scale 2", out1 => "Data_block_1"."Accumulate Scale 2")
   END_RUNG
   // the same network as SCL:
   #_w1 := "mEnableXiloFish" AND ("Data_block_1"."Set Scale 2" < "Data_block_1"."Accumulate Scale 2");
   #_w2 := #_w1 AND NOT "Tag_64";   // rising edge
   "Tag_64" := #_w1;
   IF #_w2 THEN "Data_block_1"."Accumulate Scale 2" := "Data_block_1"."Set Scale 2"; END_IF;
END_REGION

REGION Network 3
   RUNG wire#powerrail
      Contact( "mControlOn" )
      Contact( "mEnableXiloFish" )
      { S7_Templates := "SrcType := Real" } GE_Contact(in1 := "Data_block_1"."Act Scale 2", in2 := "Data_block_1"."Accumulate Scale 2")
      P_Trig( "Tag_63" )
      wire#w1
      Contact( "mEnableXiloFish13" )
      R_Coil( "mEnableXiloFish13" )
   END_RUNG
   RUNG wire#w1
      Contact( "mEnableXiloFish14" )
      R_Coil( "mEnableXiloFish14" )
   END_RUNG
   RUNG wire#w1
      Contact( "mEnableXiloFish15" )
      R_Coil( "mEnableXiloFish15" )
   END_RUNG
   RUNG wire#w1
      Contact( "mEnableXiloFish16" )
      wire#w2
      R_Coil( "mEnableXiloFish16" )
   END_RUNG
   RUNG wire#w2
      R_Coil( "mEnableXiloFish" )
   END_RUNG
   // the same network as SCL:
   #_w1 := "mControlOn" AND "mEnableXiloFish" AND ("Data_block_1"."Act Scale 2" >= "Data_block_1"."Accumulate Scale 2");
   #_w2 := #_w1 AND NOT "Tag_63";   // rising edge
   "Tag_63" := #_w1;
   IF #_w2 AND "mEnableXiloFish13" THEN "mEnableXiloFish13" := FALSE; END_IF;
   IF #_w2 AND "mEnableXiloFish14" THEN "mEnableXiloFish14" := FALSE; END_IF;
   IF #_w2 AND "mEnableXiloFish15" THEN "mEnableXiloFish15" := FALSE; END_IF;
   #_w3 := #_w2 AND "mEnableXiloFish16";
   IF #_w3 THEN
       "mEnableXiloFish16" := FALSE;
       "mEnableXiloFish" := FALSE;
   END_IF;
END_REGION

REGION Network 4
   RUNG wire#powerrail
      Contact( "mEnableXiloFish" )
      P_Trig( "Tag_65" )
      S_Coil( "mEnableXiloFish13" )
   END_RUNG
   // the same network as SCL:
   #_w1 := "mEnableXiloFish" AND NOT "Tag_65";   // rising edge
   "Tag_65" := "mEnableXiloFish";
   IF #_w1 THEN "mEnableXiloFish13" := TRUE; END_IF;
END_REGION

REGION Network 5
   RUNG wire#powerrail
      Contact( "mEnableXiloFish13" )
      N_Trig( "Tag_66" )
      S_Coil( "mEnableXiloFish14" )
   END_RUNG
   // the same network as SCL:
   #_w1 := NOT "mEnableXiloFish13" AND "Tag_66";   // falling edge
   "Tag_66" := "mEnableXiloFish13";
   IF #_w1 THEN "mEnableXiloFish14" := TRUE; END_IF;
END_REGION

REGION Network 6
   RUNG wire#powerrail
      Contact( "mEnableXiloFish14" )
      N_Trig( "Tag_67" )
      S_Coil( "mEnableXiloFish15" )
   END_RUNG
   // the same network as SCL:
   #_w1 := NOT "mEnableXiloFish14" AND "Tag_67";   // falling edge
   "Tag_67" := "mEnableXiloFish14";
   IF #_w1 THEN "mEnableXiloFish15" := TRUE; END_IF;
END_REGION

REGION Network 7
   RUNG wire#powerrail
      Contact( "mEnableXiloFish15" )
      N_Trig( "Tag_68" )
      S_Coil( "mEnableXiloFish16" )
   END_RUNG
   // the same network as SCL:
   #_w1 := NOT "mEnableXiloFish15" AND "Tag_68";   // falling edge
   "Tag_68" := "mEnableXiloFish15";
   IF #_w1 THEN "mEnableXiloFish16" := TRUE; END_IF;
END_REGION

REGION Network 8
   RUNG wire#powerrail
      Contact( "mControlOn" )
      I_Contact( "mSensorValveScale2" )
      wire#w1
      Contact( "mEnableXiloFish13" )
      Coil( "qXiloFish13" )
   END_RUNG
   RUNG wire#w1
      Contact( "mEnableXiloFish14" )
      Coil( "qXiloFish14" )
   END_RUNG
   RUNG wire#w1
      Contact( "mEnableXiloFish15" )
      Coil( "qXiloFish15" )
   END_RUNG
   RUNG wire#w1
      Contact( "mEnableXiloFish16" )
      Coil( "qXiloFish16" )
   END_RUNG
   // the same network as SCL:
   #_w1 := "mControlOn" AND NOT "mSensorValveScale2";
   "qXiloFish13" := #_w1 AND "mEnableXiloFish13";
   "qXiloFish14" := #_w1 AND "mEnableXiloFish14";
   "qXiloFish15" := #_w1 AND "mEnableXiloFish15";
   "qXiloFish16" := #_w1 AND "mEnableXiloFish16";
END_REGION
END_FUNCTION

FUNCTION "Control_MixTank" : Void   // FC12, LAD
{ S7_Optimized_Access := 'TRUE' }
VERSION : 0.1
   VAR_TEMP   // added for the SCL form of the ladder/FBD networks
      _w1 : Bool;
      _w2 : Bool;
   END_VAR
BEGIN

REGION Network 1
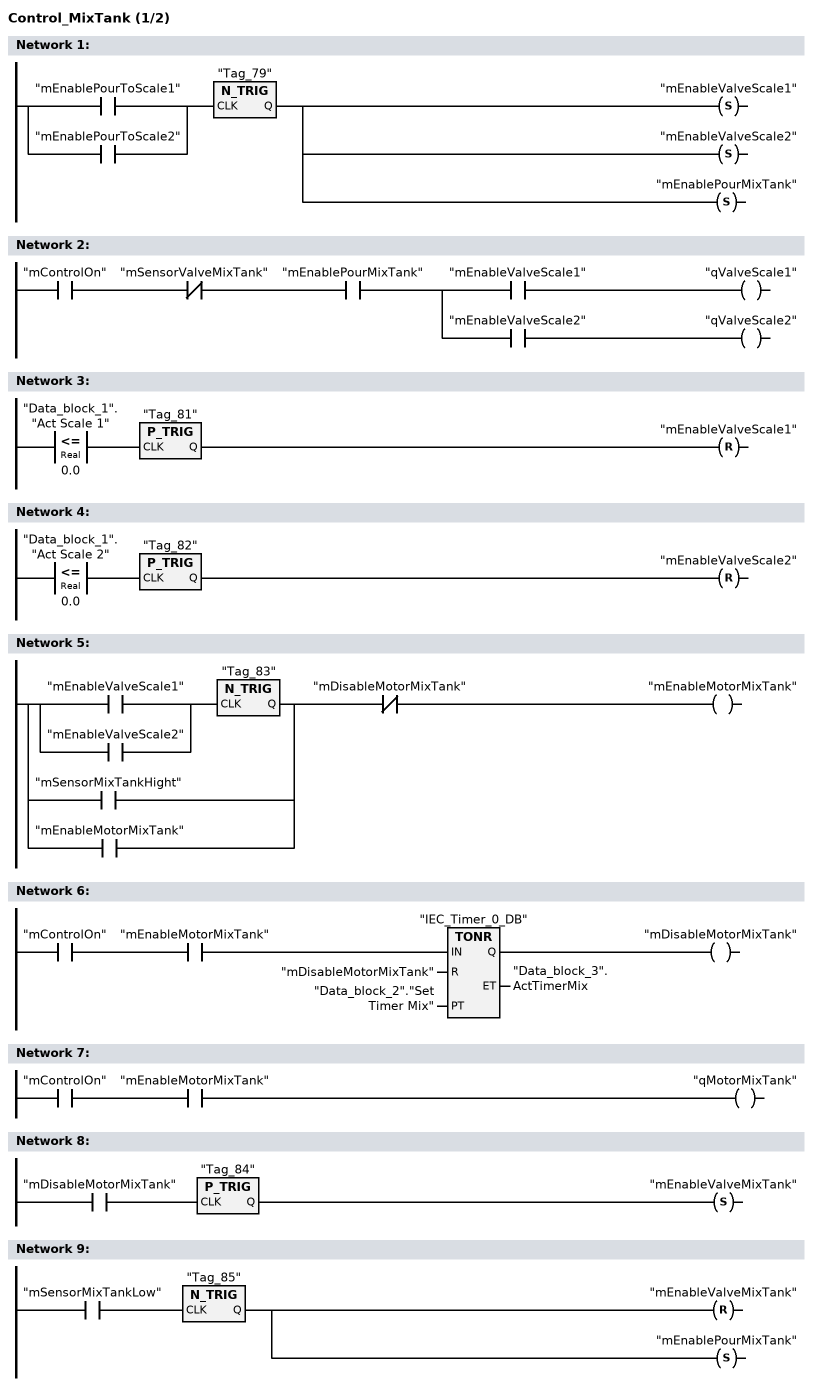
   RUNG wire#powerrail
      Contact( "mEnablePourToScale1" )
      wire#w1
      N_Trig( "Tag_79" )
      wire#w2
      S_Coil( "mEnableValveScale1" )
   END_RUNG
   RUNG wire#powerrail
      Contact( "mEnablePourToScale2" )
   END_RUNG wire#w1
   RUNG wire#w2
      S_Coil( "mEnableValveScale2" )
   END_RUNG
   RUNG wire#w2
      S_Coil( "mEnablePourMixTank" )
   END_RUNG
   // the same network as SCL:
   #_w1 := "mEnablePourToScale1" OR "mEnablePourToScale2";
   #_w2 := NOT #_w1 AND "Tag_79";   // falling edge
   "Tag_79" := #_w1;
   IF #_w2 THEN
       "mEnableValveScale1" := TRUE;
       "mEnableValveScale2" := TRUE;
       "mEnablePourMixTank" := TRUE;
   END_IF;
END_REGION

REGION Network 2
   RUNG wire#powerrail
      Contact( "mControlOn" )
      I_Contact( "mSensorValveMixTank" )
      Contact( "mEnablePourMixTank" )
      wire#w1
      Contact( "mEnableValveScale1" )
      Coil( "qValveScale1" )
   END_RUNG
   RUNG wire#w1
      Contact( "mEnableValveScale2" )
      Coil( "qValveScale2" )
   END_RUNG
   // the same network as SCL:
   #_w1 := "mControlOn" AND NOT "mSensorValveMixTank" AND "mEnablePourMixTank";
   "qValveScale1" := #_w1 AND "mEnableValveScale1";
   "qValveScale2" := #_w1 AND "mEnableValveScale2";
END_REGION

REGION Network 3
   RUNG wire#powerrail
      { S7_Templates := "SrcType := Real" } LE_Contact(in1 := "Data_block_1"."Act Scale 1", in2 := 0.0)
      P_Trig( "Tag_81" )
      R_Coil( "mEnableValveScale1" )
   END_RUNG
   // the same network as SCL:
   #_w1 := "Data_block_1"."Act Scale 1" <= 0.0;
   #_w2 := #_w1 AND NOT "Tag_81";   // rising edge
   "Tag_81" := #_w1;
   IF #_w2 THEN "mEnableValveScale1" := FALSE; END_IF;
END_REGION

REGION Network 4
   RUNG wire#powerrail
      { S7_Templates := "SrcType := Real" } LE_Contact(in1 := "Data_block_1"."Act Scale 2", in2 := 0.0)
      P_Trig( "Tag_82" )
      R_Coil( "mEnableValveScale2" )
   END_RUNG
   // the same network as SCL:
   #_w1 := "Data_block_1"."Act Scale 2" <= 0.0;
   #_w2 := #_w1 AND NOT "Tag_82";   // rising edge
   "Tag_82" := #_w1;
   IF #_w2 THEN "mEnableValveScale2" := FALSE; END_IF;
END_REGION

REGION Network 5
   RUNG wire#powerrail
      Contact( "mEnableValveScale1" )
      wire#w1
      N_Trig( "Tag_83" )
      wire#w2
      I_Contact( "mDisableMotorMixTank" )
      Coil( "mEnableMotorMixTank" )
   END_RUNG
   RUNG wire#powerrail
      Contact( "mEnableValveScale2" )
   END_RUNG wire#w1
   RUNG wire#powerrail
      Contact( "mSensorMixTankHight" )
   END_RUNG wire#w2
   RUNG wire#powerrail
      Contact( "mEnableMotorMixTank" )
   END_RUNG wire#w2
   // the same network as SCL:
   #_w1 := "mEnableValveScale1" OR "mEnableValveScale2";
   #_w2 := NOT #_w1 AND "Tag_83";   // falling edge
   "Tag_83" := #_w1;
   "mEnableMotorMixTank" := (#_w2 OR "mSensorMixTankHight" OR "mEnableMotorMixTank") AND NOT "mDisableMotorMixTank";
END_REGION

REGION Network 6
   "IEC_Timer_0_DB".TONR(IN := "mControlOn" AND "mEnableMotorMixTank",
                         R := "mDisableMotorMixTank",
                         PT := "Data_block_2"."Set Timer Mix",
                         ET => "Data_block_3".ActTimerMix);
   "mDisableMotorMixTank" := "IEC_Timer_0_DB".Q;
END_REGION

REGION Network 7
   RUNG wire#powerrail
      Contact( "mControlOn" )
      Contact( "mEnableMotorMixTank" )
      Coil( "qMotorMixTank" )
   END_RUNG
   // the same network as SCL:
   "qMotorMixTank" := "mControlOn" AND "mEnableMotorMixTank";
END_REGION

REGION Network 8
   RUNG wire#powerrail
      Contact( "mDisableMotorMixTank" )
      P_Trig( "Tag_84" )
      S_Coil( "mEnableValveMixTank" )
   END_RUNG
   // the same network as SCL:
   #_w1 := "mDisableMotorMixTank" AND NOT "Tag_84";   // rising edge
   "Tag_84" := "mDisableMotorMixTank";
   IF #_w1 THEN "mEnableValveMixTank" := TRUE; END_IF;
END_REGION

REGION Network 9
   RUNG wire#powerrail
      Contact( "mSensorMixTankLow" )
      N_Trig( "Tag_85" )
      wire#w1
      R_Coil( "mEnableValveMixTank" )
   END_RUNG
   RUNG wire#w1
      S_Coil( "mEnablePourMixTank" )
   END_RUNG
   // the same network as SCL:
   #_w1 := NOT "mSensorMixTankLow" AND "Tag_85";   // falling edge
   "Tag_85" := "mSensorMixTankLow";
   IF #_w1 THEN
       "mEnableValveMixTank" := FALSE;
       "mEnablePourMixTank" := TRUE;
   END_IF;
END_REGION

REGION Network 10
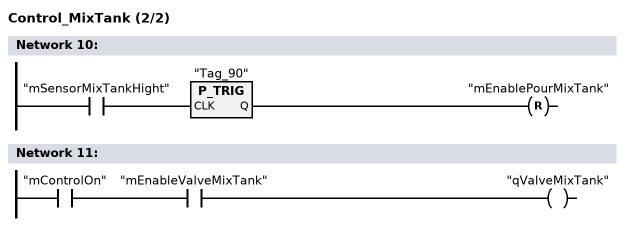
   RUNG wire#powerrail
      Contact( "mSensorMixTankHight" )
      P_Trig( "Tag_90" )
      R_Coil( "mEnablePourMixTank" )
   END_RUNG
   // the same network as SCL:
   #_w1 := "mSensorMixTankHight" AND NOT "Tag_90";   // rising edge
   "Tag_90" := "mSensorMixTankHight";
   IF #_w1 THEN "mEnablePourMixTank" := FALSE; END_IF;
END_REGION

REGION Network 11
   RUNG wire#powerrail
      Contact( "mControlOn" )
      Contact( "mEnableValveMixTank" )
      Coil( "qValveMixTank" )
   END_RUNG
   // the same network as SCL:
   "qValveMixTank" := "mControlOn" AND "mEnableValveMixTank";
END_REGION
END_FUNCTION

ORGANIZATION_BLOCK "Main"   // OB1, LAD, ProgramCycle
TITLE = "Main Program Sweep (Cycle)"
{ S7_Optimized_Access := 'TRUE' }
VERSION : 0.1
   VAR_INPUT
      Initial_Call : Bool;   // Initial call of this OB
      Remanence : Bool;   // =True, if remanent data are available
   END_VAR
BEGIN

REGION Network 1
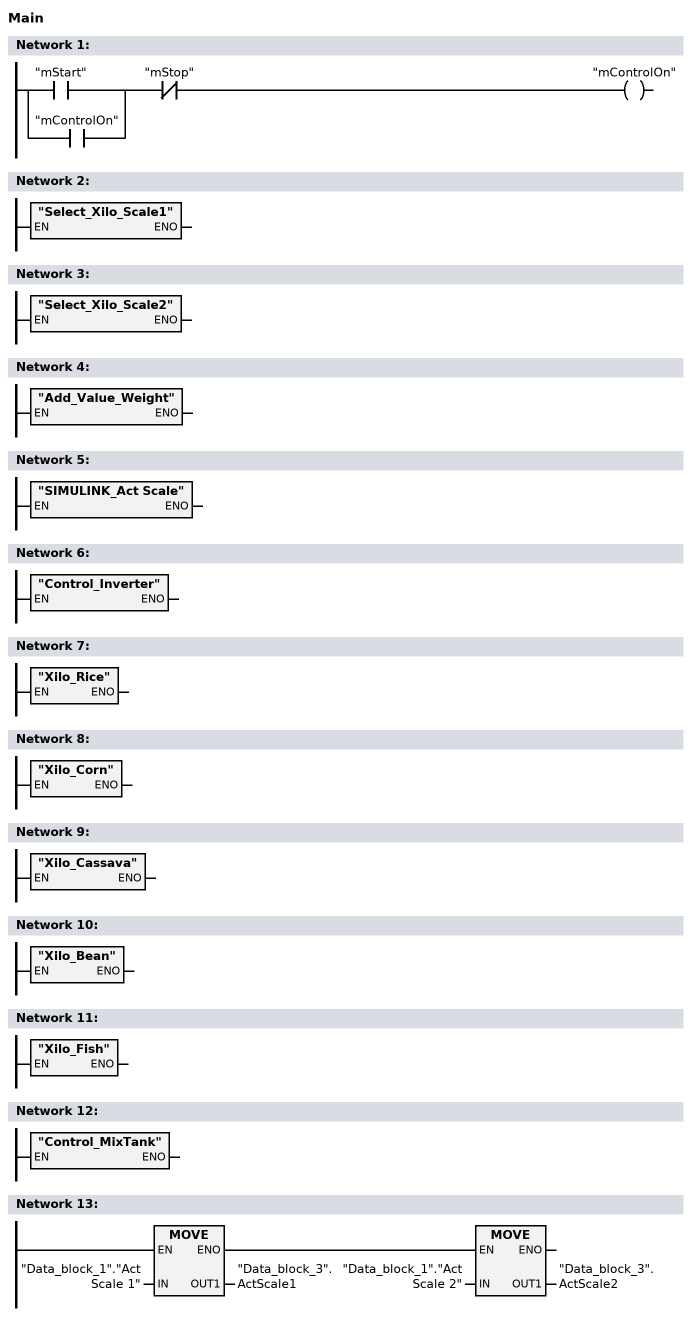
   RUNG wire#powerrail
      Contact( "mStart" )
      wire#w1
      I_Contact( "mStop" )
      Coil( "mControlOn" )
   END_RUNG
   RUNG wire#powerrail
      Contact( "mControlOn" )
   END_RUNG wire#w1
   // the same network as SCL:
   "mControlOn" := ("mStart" OR "mControlOn") AND NOT "mStop";
END_REGION

REGION Network 2
   RUNG wire#powerrail
      "Select_Xilo_Scale1"()
   END_RUNG
   // the same network as SCL:
   "Select_Xilo_Scale1"();
END_REGION

REGION Network 3
   RUNG wire#powerrail
      "Select_Xilo_Scale2"()
   END_RUNG
   // the same network as SCL:
   "Select_Xilo_Scale2"();
END_REGION

REGION Network 4
   RUNG wire#powerrail
      "Add_Value_Weight"()
   END_RUNG
   // the same network as SCL:
   "Add_Value_Weight"();
END_REGION

REGION Network 5
   RUNG wire#powerrail
      "SIMULINK_Act Scale"()
   END_RUNG
   // the same network as SCL:
   "SIMULINK_Act Scale"();
END_REGION

REGION Network 6
   RUNG wire#powerrail
      "Control_Inverter"()
   END_RUNG
   // the same network as SCL:
   "Control_Inverter"();
END_REGION

REGION Network 7
   RUNG wire#powerrail
      "Xilo_Rice"()
   END_RUNG
   // the same network as SCL:
   "Xilo_Rice"();
END_REGION

REGION Network 8
   RUNG wire#powerrail
      "Xilo_Corn"()
   END_RUNG
   // the same network as SCL:
   "Xilo_Corn"();
END_REGION

REGION Network 9
   RUNG wire#powerrail
      "Xilo_Cassava"()
   END_RUNG
   // the same network as SCL:
   "Xilo_Cassava"();
END_REGION

REGION Network 10
   RUNG wire#powerrail
      "Xilo_Bean"()
   END_RUNG
   // the same network as SCL:
   "Xilo_Bean"();
END_REGION

REGION Network 11
   RUNG wire#powerrail
      "Xilo_Fish"()
   END_RUNG
   // the same network as SCL:
   "Xilo_Fish"();
END_REGION

REGION Network 12
   RUNG wire#powerrail
      "Control_MixTank"()
   END_RUNG
   // the same network as SCL:
   "Control_MixTank"();
END_REGION

REGION Network 13
   RUNG wire#powerrail
      Move(in := "Data_block_1"."Act Scale 1", out1 => "Data_block_3".ActScale1)
      Move(in := "Data_block_1"."Act Scale 2", out1 => "Data_block_3".ActScale2)
   END_RUNG
   // the same network as SCL:
   "Data_block_3".ActScale1 := "Data_block_1"."Act Scale 1";
   "Data_block_3".ActScale2 := "Data_block_1"."Act Scale 2";
END_REGION
END_ORGANIZATION_BLOCK

(* ===== HMI "HMI_RT_1" =====
system functions are stored by id; their names below are inferred from use
connection "HMI_Connection_1": ETHERNET, S7_1200_OMS

HMI tags "Default tag table"
   "Data_block_1_Act Scale 1" : Real = PLC Data_block_1."Act Scale 1" AT %DB1.DBD20, 1 s
   "mEnablePourToScale1" : Bool = PLC mEnablePourToScale1 AT %M2.6, 1 s
   "mControlOn" : Bool = PLC mControlOn AT %M0.2, 1 s
   "mEnableXiloRice1" : Bool = PLC mEnableXiloRice1 AT %M0.4, 1 s
   "mEnableXiloRice2" : Bool = PLC mEnableXiloRice2 AT %M0.5, 1 s
   "mEnableXiloRice3" : Bool = PLC mEnableXiloRice3 AT %M0.7, 1 s
   "mEnableXiloCorn4" : Bool = PLC mEnableXiloCorn4 AT %M1.0, 1 s
   "mEnableXiloCorn5" : Bool = PLC mEnableXiloCorn5 AT %M1.1, 1 s
   "mEnableXiloCorn6" : Bool = PLC mEnableXiloCorn6 AT %M1.3, 1 s
   "mEnableXiloCorn7" : Bool = PLC mEnableXiloCorn7 AT %M1.5, 1 s
   "mEnableXiloCassava8" : Bool = PLC mEnableXiloCassava8 AT %M1.6, 1 s
   "mEnableXiloCassava9" : Bool = PLC mEnableXiloCassava9 AT %M2.0, 1 s
   "Data_block_1_Input Corn" : Real = PLC Data_block_1."Input Corn" AT %DB1.DBD4, 1 s
   "Data_block_1_Input Rice" : Real = PLC Data_block_1."Input Rice" AT %DB1.DBD0, 1 s
   "Data_block_1_Input Cassava" : Real = PLC Data_block_1."Input Cassava" AT %DB1.DBD8, 1 s
   "mEnablePourToScale2" : Bool = PLC mEnablePourToScale2 AT %M3.2, 1 s
   "mEnableXiloBean10" : Bool = PLC mEnableXiloBean10 AT %M2.1, 1 s
   "mEnableXiloBean11" : Bool = PLC mEnableXiloBean11 AT %M2.2, 1 s
   "mEnableXiloBean12" : Bool = PLC mEnableXiloBean12 AT %M3.6, 1 s
   "mEnableXiloFish13" : Bool = PLC mEnableXiloFish13 AT %M3.7, 1 s
   "mEnableXiloFish14" : Bool = PLC mEnableXiloFish14 AT %M4.0, 1 s
   "mEnableXiloFish15" : Bool = PLC mEnableXiloFish15 AT %M4.1, 1 s
   "mEnableXiloFish16" : Bool = PLC mEnableXiloFish16 AT %M4.2, 1 s
   "Data_block_1_Input Bean" : Real = PLC Data_block_1."Input Bean" AT %DB1.DBD12, 1 s
   "Data_block_1_Input Fish" : Real = PLC Data_block_1."Input Fish" AT %DB1.DBD16, 1 s
   "Data_block_1_Act Scale 2" : Real = PLC Data_block_1."Act Scale 2" AT %DB1.DBD24, 1 s

screen "Screen_1" 1920x1200
   SymbolLibrary "Symbol library_1" at 35,91 size 65x141
      Appearance <- "mEnableXiloRice1"
   SymbolLibrary "Symbol library_10" at 261,394 size 319x145
   IOField "I/O field_1" at 1761,593 size 124x37
      ProcessValue <- "Data_block_1_Act Scale 1"
   Button "Button_1" at 804,204 size 96x32; TextOff 'Scale 1'
      on Press: SetBit("mEnablePourToScale1")
      Appearance <- "mEnablePourToScale1"
   Button "Button_2" at 1564,139 size 96x32; TextOff 'On'
      on Press: SetBit("mControlOn")
      Appearance <- "mControlOn"
   SymbolLibrary "Symbol library_2" at 100,92 size 65x141
      Appearance <- "mEnableXiloRice2"
   SymbolLibrary "Symbol library_3" at 166,91 size 65x141
      Appearance <- "mEnableXiloRice3"
   SymbolLibrary "Symbol library_4" at 289,91 size 65x141
      Appearance <- "mEnableXiloCorn4"
   SymbolLibrary "Symbol library_5" at 354,91 size 65x141
      Appearance <- "mEnableXiloCorn5"
   SymbolLibrary "Symbol library_6" at 419,91 size 65x141
      Appearance <- "mEnableXiloCorn6"
   SymbolLibrary "Symbol library_7" at 484,91 size 65x141
      Appearance <- "mEnableXiloCorn7"
   SymbolLibrary "Symbol library_8" at 619,91 size 65x141
      Appearance <- "mEnableXiloCassava8"
   SymbolLibrary "Symbol library_9" at 685,92 size 65x141
      Appearance <- "mEnableXiloCassava9"
   IOField "I/O field_3" at 1761,310 size 124x37
      ProcessValue <- "Data_block_1_Input Rice"
   IOField "I/O field_2" at 1761,363 size 124x37
      ProcessValue <- "Data_block_1_Input Corn"
   IOField "I/O field_4" at 1761,423 size 124x37
      ProcessValue <- "Data_block_1_Input Cassava"
   SymbolLibrary "Symbol library_11" at 1008,392 size 319x145
   Button "Button_3" at 804,259 size 96x32; TextOff 'Scale 2'
      on Press: SetBit("mEnablePourToScale2")
      Appearance <- "mEnablePourToScale2"
   SymbolLibrary "Symbol library_12" at 943,93 size 65x141
      Appearance <- "mEnableXiloBean10"
   SymbolLibrary "Symbol library_13" at 1008,92 size 65x141
      Appearance <- "mEnableXiloBean11"
   SymbolLibrary "Symbol library_14" at 1074,92 size 65x141
      Appearance <- "mEnableXiloBean12"
   SymbolLibrary "Symbol library_15" at 1214,96 size 65x141
      Appearance <- "mEnableXiloFish13"
   SymbolLibrary "Symbol library_16" at 1279,96 size 65x141
      Appearance <- "mEnableXiloFish14"
   SymbolLibrary "Symbol library_17" at 1346,96 size 65x141
      Appearance <- "mEnableXiloFish15"
   SymbolLibrary "Symbol library_18" at 1412,96 size 65x141
      Appearance <- "mEnableXiloFish16"
   IOField "I/O field_5" at 1760,652 size 124x37
      ProcessValue <- "Data_block_1_Act Scale 2"
   IOField "I/O field_6" at 1760,480 size 124x37
      ProcessValue <- "Data_block_1_Input Bean"
   IOField "I/O field_7" at 1760,537 size 124x37
      ProcessValue <- "Data_block_1_Input Fish"
   SymbolLibrary "Symbol library_19" at 648,656 size 277x238
   Button "Button_4" at 1769,139 size 96x32; TextOff 'Off'
      on Press: SetBit("mControlOn")
      Appearance <- "mControlOn"
   TextField "Text field_1" at 1565,55 size 304x52; Text 'BẢNG ĐIỀU KHIỂN HỆ THỐNG'
   TextField "Text field_2" at 1601,233 size 222x52; Text 'THÔNG SỐ HỆ THỐNG'
   TextField "Text field_3" at 1540,316 size 99x25; Text 'Số cân gạo'
   TextField "Text field_4" at 1540,366 size 100x25; Text 'Số cân ngô'
   TextField "Text field_5" at 1540,423 size 97x25; Text 'Số cân sắn'
   TextField "Text field_6" at 1540,481 size 99x25; Text 'Số cân đậu'
   TextField "Text field_7" at 1540,542 size 86x25; Text 'Số cân cá'
   TextField "Text field_8" at 1540,597 size 161x25; Text 'Trọng lượng cân 1'
   TextField "Text field_9" at 1540,657 size 161x25; Text 'Trọng lượng cân 2'
*)